Omron Sysmac Studio project Auto Connect Project (Sysmac Studio 1.45.1.64010, StandardProject)

# Controller new_Controller_0: NX102-9000 version 1.43
Units and slaves: Node1 : NX-ECC203 (E001); Unit 1 : NX-ID5342 (N1); Unit 2 : NX-ID5342 (N2); Unit 3 : NX-OD5121 (N3); Unit 4 : NX-OD5121 (N4); Node2 : NX-ECC203 (E002); Unit 1 : NX-ID5342 (N1_1); Unit 2 : NX-ID5342 (N2_1); Unit 3 : NX-OD5121 (N3_1); Unit 4 : NX-OD5121 (N4_1); Node3 : NX-ECC203 (E003); Unit 1 : NX-ID5342 (N5); Unit 2 : NX-ID5342 (N5_2); Unit 3 : NX-OD5121 (N6); Unit 4 : NX-OD5121 (N6_1); Node4 : NX-ECC203 (E004); Unit 1 : NX-ID5342 (N1_2); Unit 2 : NX-ID5342 (N2_2); Unit 3 : NX-OD5121 (N3_2); Unit 4 : NX-OD5121 (N4_2); Node5 : NX-ECC203 (E005); Unit 1 : NX-ID5342 (N7); Unit 2 : NX-ID5342 (N7_1); Unit 3 : NX-OD5121 (N8); Unit 4 : NX-OD5121 (N8_1); Node6 : NX-ECC203 (E006); Unit 1 : NX-ID5342 (N1_3); Unit 2 : NX-ID5342 (N2_3); Unit 3 : NX-OD5121 (N3_3); Unit 4 : NX-OD5121 (N4_3); Unit 1 : NX-PF0730 (N5_1); Unit 2 : NX-OD5121 (N3_6); Unit 3 : NX-ID5342 (N2_6)
Task PrimaryTask (priority 4, period or condition 2000): Program0

VAR_GLOBAL
    IN1_00 : BOOL;  (* at ECAT://node#[1,1]/Input Bit 16 bits/Input Bit 00 *)
    IN1_01 : BOOL;  (* at ECAT://node#[1,1]/Input Bit 16 bits/Input Bit 01 *)
    IN1_02 : BOOL;  (* at ECAT://node#[1,1]/Input Bit 16 bits/Input Bit 02 *)
    IN1_03 : BOOL;  (* at ECAT://node#[1,1]/Input Bit 16 bits/Input Bit 03 *)
    IN0_01 : BOOL;  (* PB RESET; at IOBus://unit#3/Input Bit 16 bits/Input Bit 01 *)
    IN0_00 : BOOL;  (* SS ENABLE; at IOBus://unit#3/Input Bit 16 bits/Input Bit 00 *)
    OUT100_00 : BOOL;  (* PL PLC RUN; at IOBus://unit#2/Output Bit 16 bits/Output Bit 00 *)
    OUT100_01 : BOOL;  (* PL FAULT; at IOBus://unit#2/Output Bit 16 bits/Output Bit 01 *)
    OUT100_02 : BOOL;  (* PL ENABLE MODE; at IOBus://unit#2/Output Bit 16 bits/Output Bit 02 *)
    OUT100_03 : BOOL;  (* PL KUNING; at IOBus://unit#2/Output Bit 16 bits/Output Bit 03 *)
    OUT100_04 : BOOL;  (* PL KUNING; at IOBus://unit#2/Output Bit 16 bits/Output Bit 04 *)
    OUT100_05 : BOOL;  (* BUZZER; at IOBus://unit#2/Output Bit 16 bits/Output Bit 05 *)
    OUT100_06 : BOOL;  (* TL RED; at IOBus://unit#2/Output Bit 16 bits/Output Bit 06 *)
    OUT100_07 : BOOL;  (* TL YELLOW; at IOBus://unit#2/Output Bit 16 bits/Output Bit 07 *)
    OUT100_08 : BOOL;  (* TL GREEN; at IOBus://unit#2/Output Bit 16 bits/Output Bit 08 *)
    OUT101_00 : BOOL;  (* FINISH PICK RACK 1; at ECAT://node#[1,3]/Output Bit 16 bits/Output Bit 00 *)
    OUT101_01 : BOOL;  (* at ECAT://node#[1,3]/Output Bit 16 bits/Output Bit 01 *)
    OUT101_02 : BOOL;  (* at ECAT://node#[1,3]/Output Bit 16 bits/Output Bit 02 *)
    OUT101_03 : BOOL;  (* at ECAT://node#[1,3]/Output Bit 16 bits/Output Bit 03 *)
    OUT101_04 : BOOL;  (* at ECAT://node#[1,3]/Output Bit 16 bits/Output Bit 04 *)
    OUT102_00 : BOOL;  (* at ECAT://node#[1,4]/Output Bit 16 bits/Output Bit 00 *)
    OUT103_00 : BOOL;  (* FINISH PICK RACK 2; at ECAT://node#[2,3]/Output Bit 16 bits/Output Bit 00 *)
    OUT103_01 : BOOL;  (* at ECAT://node#[2,3]/Output Bit 16 bits/Output Bit 01 *)
    OUT103_02 : BOOL;  (* at ECAT://node#[2,3]/Output Bit 16 bits/Output Bit 02 *)
    OUT103_03 : BOOL;  (* at ECAT://node#[2,3]/Output Bit 16 bits/Output Bit 03 *)
    OUT103_04 : BOOL;  (* at ECAT://node#[2,3]/Output Bit 16 bits/Output Bit 04 *)
    OUT103_05 : BOOL;  (* at ECAT://node#[2,3]/Output Bit 16 bits/Output Bit 05 *)
    OUT103_06 : BOOL;  (* at ECAT://node#[2,3]/Output Bit 16 bits/Output Bit 06 *)
    OUT103_07 : BOOL;  (* at ECAT://node#[2,3]/Output Bit 16 bits/Output Bit 07 *)
    OUT103_08 : BOOL;  (* at ECAT://node#[2,3]/Output Bit 16 bits/Output Bit 08 *)
    OUT103_09 : BOOL;  (* at ECAT://node#[2,3]/Output Bit 16 bits/Output Bit 09 *)
    OUT103_10 : BOOL;  (* at ECAT://node#[2,3]/Output Bit 16 bits/Output Bit 10 *)
    OUT104_00 : BOOL;  (* at ECAT://node#[2,4]/Output Bit 16 bits/Output Bit 00 *)
    OUT107_00 : BOOL;  (* at ECAT://node#[4,3]/Output Bit 16 bits/Output Bit 00 *)
    OUT107_01 : BOOL;  (* at ECAT://node#[4,3]/Output Bit 16 bits/Output Bit 01 *)
    OUT107_02 : BOOL;  (* at ECAT://node#[4,3]/Output Bit 16 bits/Output Bit 02 *)
    OUT107_03 : BOOL;  (* at ECAT://node#[4,3]/Output Bit 16 bits/Output Bit 03 *)
    OUT107_04 : BOOL;  (* at ECAT://node#[4,3]/Output Bit 16 bits/Output Bit 04 *)
    OUT107_05 : BOOL;  (* at ECAT://node#[4,3]/Output Bit 16 bits/Output Bit 05 *)
    OUT107_06 : BOOL;  (* at ECAT://node#[4,3]/Output Bit 16 bits/Output Bit 06 *)
    OUT107_07 : BOOL;  (* at ECAT://node#[4,3]/Output Bit 16 bits/Output Bit 07 *)
    OUT107_09 : BOOL;  (* at ECAT://node#[4,3]/Output Bit 16 bits/Output Bit 09 *)
    OUT107_10 : BOOL;  (* at ECAT://node#[4,3]/Output Bit 16 bits/Output Bit 10 *)
    OUT107_11 : BOOL;  (* at ECAT://node#[4,3]/Output Bit 16 bits/Output Bit 11 *)
    OUT107_12 : BOOL;  (* at ECAT://node#[4,3]/Output Bit 16 bits/Output Bit 12 *)
    OUT107_13 : BOOL;  (* at ECAT://node#[4,3]/Output Bit 16 bits/Output Bit 13 *)
    OUT107_14 : BOOL;  (* at ECAT://node#[4,3]/Output Bit 16 bits/Output Bit 14 *)
    OUT108_15 : BOOL;  (* at ECAT://node#[4,4]/Output Bit 16 bits/Output Bit 15 *)
    OUT111_01 : BOOL;  (* at ECAT://node#[6,3]/Output Bit 16 bits/Output Bit 01 *)
    OUT111_02 : BOOL;  (* at ECAT://node#[6,3]/Output Bit 16 bits/Output Bit 02 *)
    OUT112_00 : BOOL;  (* at ECAT://node#[6,4]/Output Bit 16 bits/Output Bit 00 *)
    OUT112_01 : BOOL;  (* at ECAT://node#[6,4]/Output Bit 16 bits/Output Bit 01 *)
    IN1_08 : BOOL;  (* at ECAT://node#[1,1]/Input Bit 16 bits/Input Bit 08 *)
    IN2_15 : BOOL;  (* at ECAT://node#[1,2]/Input Bit 16 bits/Input Bit 15 *)
    IN3_00 : BOOL;  (* at ECAT://node#[2,1]/Input Bit 16 bits/Input Bit 00 *)
    IN3_01 : BOOL;  (* at ECAT://node#[2,1]/Input Bit 16 bits/Input Bit 01 *)
    IN3_02 : BOOL;  (* at ECAT://node#[2,1]/Input Bit 16 bits/Input Bit 02 *)
    IN3_03 : BOOL;  (* at ECAT://node#[2,1]/Input Bit 16 bits/Input Bit 03 *)
    IN3_04 : BOOL;  (* at ECAT://node#[2,1]/Input Bit 16 bits/Input Bit 04 *)
    IN3_05 : BOOL;  (* at ECAT://node#[2,1]/Input Bit 16 bits/Input Bit 05 *)
    IN3_06 : BOOL;  (* at ECAT://node#[2,1]/Input Bit 16 bits/Input Bit 06 *)
    IN3_07 : BOOL;  (* at ECAT://node#[2,1]/Input Bit 16 bits/Input Bit 07 *)
    IN3_08 : BOOL;  (* at ECAT://node#[2,1]/Input Bit 16 bits/Input Bit 08 *)
    IN3_09 : BOOL;  (* at ECAT://node#[2,1]/Input Bit 16 bits/Input Bit 09 *)
    IN7_01 : BOOL;  (* at ECAT://node#[4,1]/Input Bit 16 bits/Input Bit 01 *)
    IN7_02 : BOOL;  (* at ECAT://node#[4,1]/Input Bit 16 bits/Input Bit 02 *)
    IN7_03 : BOOL;  (* at ECAT://node#[4,1]/Input Bit 16 bits/Input Bit 03 *)
    IN7_04 : BOOL;  (* at ECAT://node#[4,1]/Input Bit 16 bits/Input Bit 04 *)
    IN7_05 : BOOL;  (* at ECAT://node#[4,1]/Input Bit 16 bits/Input Bit 05 *)
    IN7_06 : BOOL;  (* at ECAT://node#[4,1]/Input Bit 16 bits/Input Bit 06 *)
    IN7_07 : BOOL;  (* at ECAT://node#[4,1]/Input Bit 16 bits/Input Bit 07 *)
    IN7_09 : BOOL;  (* at ECAT://node#[4,1]/Input Bit 16 bits/Input Bit 09 *)
    IN7_10 : BOOL;  (* at ECAT://node#[4,1]/Input Bit 16 bits/Input Bit 10 *)
    IN7_11 : BOOL;  (* at ECAT://node#[4,1]/Input Bit 16 bits/Input Bit 11 *)
    IN7_12 : BOOL;  (* at ECAT://node#[4,1]/Input Bit 16 bits/Input Bit 12 *)
    IN7_13 : BOOL;  (* at ECAT://node#[4,1]/Input Bit 16 bits/Input Bit 13 *)
    IN7_14 : BOOL;  (* at ECAT://node#[4,1]/Input Bit 16 bits/Input Bit 14 *)
    IN11_01 : BOOL;  (* at ECAT://node#[6,1]/Input Bit 16 bits/Input Bit 01 *)
    IN11_02 : BOOL;  (* at ECAT://node#[6,1]/Input Bit 16 bits/Input Bit 02 *)
    IN7_00 : BOOL;  (* at ECAT://node#[4,1]/Input Bit 16 bits/Input Bit 00 *)
    ATCO_NICKEL : BOOL;
    ATCO_LITHIUM : BOOL;
    NEW_BATTERY : BOOL;
    DATA_ATCO : WORD;  (* Area Loading *)
    PLC_ERROR_CODE : DWORD;
    OLD_DATA_ATCO : WORD;
    SEN_RACK1A_UP1 AT %W31.00 : BOOL;  (* published *)
    SEN_RACK1A_MD1 AT %W31.01 : BOOL;  (* published *)
    SEN_RACK1A_LO1 AT %W31.06 : BOOL;  (* published *)
    SEN_RACK1B_UP1 AT %W31.02 : BOOL;  (* published *)
    SEN_RACK1B_UP2 AT %W31.03 : BOOL;  (* published *)
    SEN_RACK1B_UP3 AT %W31.04 : BOOL;  (* published *)
    SEN_RACK1B_MD1 AT %W31.05 : BOOL;  (* published *)
    SEN_RACK1B_LO1 AT %W31.07 : BOOL;  (* published *)
    LAMP_RACK1A_UP1 AT %W21.00 : BOOL;  (* published *)
    LAMP_RACK1A_MD1 AT %W21.01 : BOOL;  (* published *)
    LAMP_RACK1A_LO1 AT %W21.06 : BOOL;  (* published *)
    LAMP_RACK1B_UP1 AT %W21.02 : BOOL;  (* published *)
    LAMP_RACK1B_UP2 AT %W21.03 : BOOL;  (* published *)
    LAMP_RACK1B_UP3 AT %W21.04 : BOOL;  (* published *)
    LAMP_RACK1B_MD1 AT %W21.05 : BOOL;  (* published *)
    LAMP_RACK1B_LO1 AT %W21.07 : BOOL;  (* published *)
    SEN_RACK2A_UP1 AT %W32.00 : BOOL;  (* published *)
    SEN_RACK2A_UP2 AT %W32.01 : BOOL;  (* published *)
    SEN_RACK2A_MD1 AT %W32.02 : BOOL;  (* published *)
    SEN_RACK2A_MD2 AT %W32.03 : BOOL;  (* published *)
    SEN_RACK2B_UP1 AT %W32.04 : BOOL;  (* published *)
    SEN_RACK2B_UP2 AT %W32.05 : BOOL;  (* published *)
    SEN_RACK2B_MD1 AT %W32.06 : BOOL;  (* published *)
    SEN_RACK2B_MD2 AT %W32.07 : BOOL;  (* published *)
    SEN_RACK2B_LO1 AT %W32.08 : BOOL;  (* published *)
    SEN_RACK2B_LO2 AT %W32.09 : BOOL;  (* published *)
    LAMP_RACK2A_UP1 AT %W22.00 : BOOL;  (* published *)
    LAMP_RACK2A_UP2 AT %W22.01 : BOOL;  (* published *)
    LAMP_RACK2A_MD1 AT %W22.02 : BOOL;  (* published *)
    LAMP_RACK2A_MD2 AT %W22.03 : BOOL;  (* published *)
    LAMP_RACK2B_UP1 AT %W22.04 : BOOL;  (* published *)
    LAMP_RACK2B_UP2 AT %W22.05 : BOOL;  (* published *)
    LAMP_RACK2B_MD1 AT %W22.06 : BOOL;  (* published *)
    LAMP_RACK2B_MD2 AT %W22.07 : BOOL;  (* published *)
    LAMP_RACK2B_LO1 AT %W22.08 : BOOL;  (* published *)
    LAMP_RACK2B_LO2 AT %W22.09 : BOOL;  (* published *)
    SEN_RACK3A_UP1 AT %W33.00 : BOOL;  (* published *)
    SEN_RACK3A_MD1 AT %W33.01 : BOOL;  (* published *)
    LAMP_RACK3A_UP1 AT %W23.00 : BOOL;  (* published *)
    LAMP_RACK3A_MD1 AT %W23.01 : BOOL;  (* published *)
    SEN_RACK4A_UP1 AT %W34.00 : BOOL;  (* published *)
    SEN_RACK4A_UP2 AT %W34.01 : BOOL;  (* published *)
    SEN_RACK4A_MD1 AT %W34.02 : BOOL;  (* published *)
    SEN_RACK4A_MD2 AT %W34.03 : BOOL;  (* published *)
    SEN_RACK4A_MD3 AT %W34.04 : BOOL;  (* published *)
    SEN_RACK4A_LO1 AT %W34.05 : BOOL;  (* published *)
    SEN_RACK4A_LO2 AT %W34.06 : BOOL;  (* published *)
    SEN_RACK4A_LO3 AT %W34.07 : BOOL;  (* published *)
    SEN_RACK4B_UP1 AT %W34.08 : BOOL;  (* published *)
    SEN_RACK4B_MD1 AT %W34.09 : BOOL;  (* published *)
    SEN_RACK4B_MD2 AT %W34.10 : BOOL;  (* published *)
    SEN_RACK4B_LO1 AT %W34.11 : BOOL;  (* published *)
    SEN_RACK4B_LO2 AT %W34.12 : BOOL;  (* published *)
    SEN_RACK4C_UP1 AT %W34.13 : BOOL;  (* published *)
    SEN_RACK4C_MD1 AT %W34.14 : BOOL;  (* published *)
    SEN_RACK4C_LO1 AT %W34.15 : BOOL;  (* published *)
    LAMP_RACK4A_UP1 AT %W24.00 : BOOL;  (* published *)
    LAMP_RACK4A_UP2 AT %W24.01 : BOOL;  (* published *)
    LAMP_RACK4A_MD1 AT %W24.02 : BOOL;  (* published *)
    LAMP_RACK4A_MD2 AT %W24.03 : BOOL;  (* published *)
    LAMP_RACK4A_MD3 AT %W24.04 : BOOL;  (* published *)
    LAMP_RACK4A_LO1 AT %W24.05 : BOOL;  (* published *)
    LAMP_RACK4A_LO2 AT %W24.06 : BOOL;  (* published *)
    LAMP_RACK4A_LO3 AT %W24.07 : BOOL;  (* published *)
    LAMP_RACK4B_UP1 AT %W24.08 : BOOL;  (* published *)
    LAMP_RACK4B_MD1 AT %W24.09 : BOOL;  (* published *)
    LAMP_RACK4B_MD2 AT %W24.10 : BOOL;  (* published *)
    LAMP_RACK4B_LO1 AT %W24.11 : BOOL;  (* published *)
    LAMP_RACK4B_LO2 AT %W24.12 : BOOL;  (* published *)
    LAMP_RACK4C_UP1 AT %W24.13 : BOOL;  (* published *)
    LAMP_RACK4C_MD1 AT %W24.14 : BOOL;  (* published *)
    LAMP_RACK4C_LO1 AT %W24.15 : BOOL;  (* published *)
    SEN_RACK5A_UP1 AT %W35.00 : BOOL;  (* published *)
    SEN_RACK5A_MD1 AT %W35.01 : BOOL;  (* published *)
    SEN_RACK5A_LO1 AT %W35.02 : BOOL;  (* published *)
    SEN_RACK5B_UP1 AT %W35.03 : BOOL;  (* published *)
    SEN_RACK5B_MD1 AT %W35.04 : BOOL;  (* published *)
    SEN_RACK5B_LO1 AT %W35.05 : BOOL;  (* published *)
    LAMP_RACK5A_UP1 AT %W25.00 : BOOL;  (* published *)
    LAMP_RACK5A_MD1 AT %W25.01 : BOOL;  (* published *)
    LAMP_RACK5A_LO1 AT %W25.02 : BOOL;  (* published *)
    LAMP_RACK5B_UP1 AT %W25.03 : BOOL;  (* published *)
    LAMP_RACK5B_MD1 AT %W25.04 : BOOL;  (* published *)
    LAMP_RACK5B_LO1 AT %W25.05 : BOOL;  (* published *)
    SEN_RACK6A_UP1 AT %W36.00 : BOOL;  (* published *)
    SEN_RACK6A_MD1 AT %W36.01 : BOOL;  (* published *)
    SEN_RACK6A_LO1 AT %W36.02 : BOOL;  (* published *)
    SEN_RACK6B_UP1 AT %W36.03 : BOOL;  (* published *)
    SEN_RACK6B_MD1 AT %W36.05 : BOOL;  (* published *)
    LAMP_RACK6A_UP1 AT %W26.00 : BOOL;  (* published *)
    LAMP_RACK6A_MD1 AT %W26.01 : BOOL;  (* published *)
    LAMP_RACK6A_LO1 AT %W26.02 : BOOL;  (* published *)
    LAMP_RACK6B_UP1 AT %W26.03 : BOOL;  (* published *)
    LAMP_RACK6B_MD1 AT %W26.05 : BOOL;  (* published *)
    SEN_RACK7A_UP1 AT %W37.00 : BOOL;  (* published *)
    SEN_RACK7B_UP1 AT %W37.01 : BOOL;  (* published *)
END_VAR
VAR_GLOBAL RETAIN
    TEACH_RACK1A_LO1 : WORD;
    TEACH_RACK1A_MD1 : WORD;
    TEACH_RACK1A_UP1 : WORD;
    TEACH_RACK1B_LO1 : WORD;
    TEACH_RACK1B_MD1 : WORD;
    TEACH_RACK1B_UP1 : WORD;
    TEACH_RACK1B_UP2 : WORD;
    TEACH_RACK1B_UP3 : WORD;
    TEACH_RACK2A_MD1 : WORD;
    TEACH_RACK2A_MD2 : WORD;
    TEACH_RACK2A_UP1 : WORD;
    TEACH_RACK2A_UP2 : WORD;
    TEACH_RACK2B_LO1 : WORD;
    TEACH_RACK2B_LO2 : WORD;
    TEACH_RACK2B_MD1 : WORD;
    TEACH_RACK2B_MD2 : WORD;
    TEACH_RACK2B_UP1 : WORD;
    TEACH_RACK2B_UP2 : WORD;
    TEACH_RACK3A_MD1 : WORD;
    TEACH_RACK3A_UP1 : WORD;
    TEACH_RACK4A_LO1 : WORD;
    TEACH_RACK4A_LO2 : WORD;
    TEACH_RACK4A_LO3 : WORD;
    TEACH_RACK4A_MD1 : WORD;
    TEACH_RACK4A_MD2 : WORD;
    TEACH_RACK4A_MD3 : WORD;
    TEACH_RACK4A_UP1 : WORD;
    TEACH_RACK4A_UP2 : WORD;
    TEACH_RACK4B_LO1 : WORD;
    TEACH_RACK4B_LO2 : WORD;
    TEACH_RACK4B_MD1 : WORD;
    TEACH_RACK4B_MD2 : WORD;
    TEACH_RACK4B_UP1 : WORD;
    TEACH_RACK4C_LO1 : WORD;
    TEACH_RACK4C_MD1 : WORD;
    TEACH_RACK4C_UP1 : WORD;
    TEACH_RACK5A_LO1 : WORD;
    TEACH_RACK5A_MD1 : WORD;
    TEACH_RACK5A_UP1 : WORD;
    TEACH_RACK5B_LO1 : WORD;
    TEACH_RACK5B_MD1 : WORD;
    TEACH_RACK5B_UP1 : WORD;
    TEACH_RACK6A_LO1 : WORD;
    TEACH_RACK6A_MD1 : WORD;
    TEACH_RACK6A_UP1 : WORD;
    TEACH_RACK6B_MD1 : WORD;
    TEACH_RACK6B_UP1 : WORD;
    TEACH_RACK7A_UP1 : WORD;
END_VAR
VAR_GLOBAL
    LAMP_RACK7A_UP1 AT %W27.00 : BOOL;  (* published *)
    LAMP_RACK7B_UP1 AT %W27.01 : BOOL;  (* published *)
    FINISH_PICK_RACK1 : BOOL;
    FINISH_PICK_RACK2 : BOOL;
    FINISH_PICK_RACK4 : BOOL;
    FINISH_PICK_RACK6 : BOOL;
    FINISH_PICK_RACK7 : BOOL;
    FAULT_PICK_FALSE_RACK1 : BOOL;
    FAULT_PICK_FALSE_RACK2 : BOOL;
    FAULT_PICK_FALSE_RACK4 : BOOL;
    FAULT_PICK_FALSE_RACK6 : BOOL;
    FAULT_PICK_FALSE_RACK7 : BOOL;
    FAULT_PICK_TOO_MUCH_RACK1 : BOOL;
    FAULT_PICK_TOO_MUCH_RACK2 : BOOL;
    FAULT_PICK_TOO_MUCH_RACK4 : BOOL;
    FAULT_PICK_TOO_MUCH_RACK6 : BOOL;
    FAULT_PICK_TOO_MUCH_RACK7 : BOOL;
END_VAR
VAR_GLOBAL RETAIN
    TEACH_RACK7B_UP1 : WORD;
END_VAR
VAR_GLOBAL
    ATCO_UDP_CONNECTED : BOOL;
    DATA_ATCO_1 : WORD;  (* Area Lower Case *)
    DATA_ATCO_2 : WORD;  (* Area BBM *)
    DATA_ATCO_3 : WORD;  (* Area Manual Tightening *)
    DATA_ATCO_4 : WORD;  (* Area Charging *)
    ATCO_NICKEL_1 : BOOL;
    ATCO_LITHIUM_1 : BOOL;
    NEW_BATTERY_1 : BOOL;
    ATCO_NICKEL_2 : BOOL;
    ATCO_LITHIUM_2 : BOOL;
    NEW_BATTERY_2 : BOOL;
    ATCO_NICKEL_3 : BOOL;
    ATCO_LITHIUM_3 : BOOL;
    NEW_BATTERY_3 : BOOL;
    ATCO_NICKEL_4 : BOOL;
    ATCO_LITHIUM_4 : BOOL;
    NEW_BATTERY_4 : BOOL;
    FLAG_ERROR_PICK : BOOL;
END_VAR
VAR_GLOBAL RETAIN
    HMI_SET_1A_UP1 AT %D0 : INT;  (* published *)
    HMI_SET_1A_MD1 AT %D1 : INT;  (* published *)
    HMI_SET_1B_UP1 AT %D2 : INT;  (* published *)
    HMI_SET_1B_UP2 AT %D3 : INT;  (* published *)
    HMI_SET_1B_UP3 AT %D4 : INT;  (* published *)
    HMI_SET_1B_MD1 AT %D5 : INT;  (* published *)
    HMI_SET_2A_UP1 AT %D6 : INT;  (* published *)
    HMI_SET_2A_UP2 AT %D7 : INT;  (* published *)
    HMI_SET_2A_MD1 AT %D8 : INT;  (* published *)
    HMI_SET_2A_MD2 AT %D9 : INT;  (* published *)
    HMI_SET_2B_UP1 AT %D10 : INT;  (* published *)
    HMI_SET_2B_UP2 AT %D11 : INT;  (* published *)
    HMI_SET_2B_MD1 AT %D12 : INT;  (* published *)
    HMI_SET_2B_MD2 AT %D13 : INT;  (* published *)
    HMI_SET_2B_LO1 AT %D14 : INT;  (* published *)
    HMI_SET_2B_LO2 AT %D15 : INT;  (* published *)
    HMI_SET_3A_UP1 AT %D16 : INT;  (* published *)
    HMI_SET_3A_MD1 AT %D17 : INT;  (* published *)
    HMI_SET_4A_UP1 AT %D18 : INT;  (* published *)
    HMI_SET_4A_UP2 AT %D19 : INT;  (* published *)
    HMI_SET_4A_MD1 AT %D20 : INT;  (* published *)
    HMI_SET_4A_MD2 AT %D21 : INT;  (* published *)
    HMI_SET_4A_MD3 AT %D22 : INT;  (* published *)
    HMI_SET_4A_LO1 AT %D23 : INT;  (* published *)
    HMI_SET_4A_LO2 AT %D24 : INT;  (* published *)
    HMI_SET_4A_LO3 AT %D25 : INT;  (* published *)
    HMI_SET_4B_UP1 AT %D26 : INT;  (* published *)
    HMI_SET_4B_MD1 AT %D27 : INT;  (* published *)
    HMI_SET_4B_MD2 AT %D28 : INT;  (* published *)
    HMI_SET_4B_LO1 AT %D29 : INT;  (* published *)
    HMI_SET_4B_LO2 AT %D30 : INT;  (* published *)
    HMI_SET_4C_UP1 AT %D31 : INT;  (* published *)
    HMI_SET_4C_MD1 AT %D32 : INT;  (* published *)
    HMI_SET_4C_LO1 AT %D33 : INT;  (* published *)
    HMI_SET_5A_UP1 AT %D34 : INT;  (* published *)
    HMI_SET_5A_MD1 AT %D35 : INT;  (* published *)
    HMI_SET_5A_LO1 AT %D36 : INT;  (* published *)
    HMI_SET_5B_UP1 AT %D37 : INT;  (* published *)
    HMI_SET_5B_MD1 AT %D38 : INT;  (* published *)
    HMI_SET_6A_UP1 AT %D39 : INT;  (* published *)
    HMI_SET_6A_MD1 AT %D40 : INT;  (* published *)
    HMI_SET_6A_LO1 AT %D41 : INT;  (* published *)
    HMI_SET_6B_UP1 AT %D42 : INT;  (* published *)
    HMI_SET_6B_UP2 AT %D43 : INT;  (* published *)
    HMI_SET_6B_MD1 AT %D44 : INT;  (* published *)
END_VAR
VAR_GLOBAL
    HMI_POWER_ON AT %W0.08 : BOOL;  (* published *)
    HMI_ENABLE AT %W0.01 : BOOL;  (* published *)
    HMI_CONNECT AT %W0.02 : BOOL;  (* published *)
    HMI_NICKEL_BATTERY AT %W0.03 : BOOL;  (* published *)
    HMI_LITHIUM_BATTERY AT %W0.04 : BOOL;  (* published *)
    HMI_PLC_RUN AT %W0.05 : BOOL;  (* published *)
    HMI_FAULT AT %W0.06 : BOOL;  (* published *)
    HMI_ENABLE_SETTING AT %W0.07 : BOOL;  (* published *)
    HMI_LAMPU_1A_UP1 AT %W1.00 : BOOL;  (* published *)
    HMI_LAMPU_1A_MD1 AT %W1.01 : BOOL;  (* published *)
    HMI_LAMPU_1B_UP1 AT %W1.02 : BOOL;  (* published *)
    HMI_LAMPU_1B_UP2 AT %W1.03 : BOOL;  (* published *)
    HMI_LAMPU_1B_UP3 AT %W1.04 : BOOL;  (* published *)
    HMI_LAMPU_1B_MD1 AT %W1.05 : BOOL;  (* published *)
    HMI_LAMPU_2A_UP1 AT %W2.00 : BOOL;  (* published *)
    HMI_LAMPU_2A_UP2 AT %W2.01 : BOOL;  (* published *)
    HMI_LAMPU_2A_MD1 AT %W2.02 : BOOL;  (* published *)
    HMI_LAMPU_2A_MD2 AT %W2.03 : BOOL;  (* published *)
    HMI_LAMPU_2B_UP1 AT %W2.04 : BOOL;  (* published *)
    HMI_LAMPU_2B_UP2 AT %W2.05 : BOOL;  (* published *)
    HMI_LAMPU_2B_MD1 AT %W2.06 : BOOL;  (* published *)
    HMI_LAMPU_2B_MD2 AT %W2.07 : BOOL;  (* published *)
    HMI_LAMPU_2B_LO1 AT %W2.08 : BOOL;  (* published *)
    HMI_LAMPU_2B_LO2 AT %W2.09 : BOOL;  (* published *)
    HMI_LAMPU_3A_UP1 AT %W3.00 : BOOL;  (* published *)
    HMI_LAMPU_3A_MD1 AT %W3.01 : BOOL;  (* published *)
    HMI_LAMPU_4A_UP1 AT %W4.00 : BOOL;  (* published *)
    HMI_LAMPU_4A_UP2 AT %W4.01 : BOOL;  (* published *)
    HMI_LAMPU_4A_MD1 AT %W4.02 : BOOL;  (* published *)
    HMI_LAMPU_4A_MD2 AT %W4.03 : BOOL;  (* published *)
    HMI_LAMPU_4A_MD3 AT %W4.04 : BOOL;  (* published *)
    HMI_LAMPU_4A_LO1 AT %W4.05 : BOOL;  (* published *)
    HMI_LAMPU_4A_LO2 AT %W4.06 : BOOL;  (* published *)
    HMI_LAMPU_4A_LO3 AT %W4.07 : BOOL;  (* published *)
    HMI_LAMPU_4B_UP1 AT %W4.08 : BOOL;  (* published *)
    HMI_LAMPU_4B_MD1 AT %W4.09 : BOOL;  (* published *)
    HMI_LAMPU_4B_MD2 AT %W4.10 : BOOL;  (* published *)
    HMI_LAMPU_4B_LO1 AT %W4.11 : BOOL;  (* published *)
    HMI_LAMPU_4B_LO2 AT %W4.12 : BOOL;  (* published *)
    HMI_LAMPU_4C_UP1 AT %W4.13 : BOOL;  (* published *)
    HMI_LAMPU_4C_MD1 AT %W4.14 : BOOL;  (* published *)
    HMI_LAMPU_4C_LO1 AT %W4.15 : BOOL;  (* published *)
    HMI_LAMPU_5A_UP1 AT %W5.00 : BOOL;  (* published *)
    HMI_LAMPU_5A_MD1 AT %W5.01 : BOOL;  (* published *)
    HMI_LAMPU_5A_LO1 AT %W5.02 : BOOL;  (* published *)
    HMI_LAMPU_5B_UP1 AT %W5.03 : BOOL;  (* published *)
    HMI_LAMPU_5B_MD1 AT %W5.04 : BOOL;  (* published *)
    HMI_LAMPU_6A_UP1 AT %W6.00 : BOOL;  (* published *)
    HMI_LAMPU_6A_MD1 AT %W6.01 : BOOL;  (* published *)
    HMI_LAMPU_6A_LO1 AT %W6.02 : BOOL;  (* published *)
    HMI_LAMPU_6B_UP1 AT %W6.03 : BOOL;  (* published *)
    HMI_LAMPU_6B_UP2 AT %W6.04 : BOOL;  (* published *)
    HMI_LAMPU_6B_MD1 AT %W6.05 : BOOL;  (* published *)
END_VAR
VAR_GLOBAL RETAIN
    TEACH_RACK6B_UP2 : WORD;
END_VAR
VAR_GLOBAL
    RECIEVECJ_DONE : BOOL;
    HMI_LAMPU_1A_UP2 AT %W1.06 : BOOL;  (* published *)
    HMI_LAMPU_1A_UP3 AT %W1.07 : BOOL;  (* published *)
    HMI_LAMPU_3A_UP2 AT %W3.02 : BOOL;  (* published *)
    HMI_LAMPU_3A_UP3 AT %W3.03 : BOOL;  (* published *)
    HMI_LAMPU_3A_MD2 AT %W3.04 : BOOL;  (* published *)
    HMI_LAMPU_7A_UP1 AT %W7.00 : BOOL;
    HMI_LAMPU_7A_UP2 AT %W7.01 : BOOL;
END_VAR
VAR_GLOBAL RETAIN
    HMI_SET_7A_UP1 AT %D45 : INT;  (* published *)
    HMI_SET_7A_UP2 AT %D46 : INT;  (* published *)
    HMI_SET_3A_UP2 AT %D47 : INT;  (* published *)
    HMI_SET_3A_UP3 AT %D48 : INT;  (* published *)
    HMI_SET_3A_MD2 AT %D49 : INT;  (* published *)
    HMI_SET_1A_UP2 AT %D50 : INT;  (* published *)
    HMI_SET_1A_UP3 AT %D51 : INT;  (* published *)
END_VAR
VAR_GLOBAL
    HMI_BATTERY_SETTING AT %W0.00 : BOOL;  (* published *)
    WAIT_ALARM : BOOL;
    BUZZER_OFF AT %W0.09 : BOOL;  (* published *)
END_VAR
VAR_GLOBAL RETAIN
    RAK_1_CONDITION AT %D47 : INT;  (* published *)
    RAK_2_CONDITION AT %D48 : INT;  (* published *)
    RAK_3_CONDITION AT %D49 : INT;  (* published *)
    RAK_4_CONDITION AT %D50 : INT;  (* published *)
    RAK_5_CONDITION AT %D51 : INT;  (* published *)
    RAK_6_CONDITION AT %D52 : INT;  (* published *)
    RAK_7_CONDITION AT %D53 : INT;  (* published *)
END_VAR
VAR_GLOBAL
    HMI_FAULT_PICKING AT %W0.10 : BOOL;  (* published *)
    HMI_FAULT_WAIT_PICKING AT %W0.11 : BOOL;  (* published *)
    HMI_FAULT_CONNECTION AT %W0.12 : BOOL;  (* published *)
    PROX_SUB_CONVEYOR_1 : BOOL;
    HMI_RESET_CJ AT %W0.13 : BOOL;  (* published *)
    HMI_FORCE_RAK_1 AT %W10.00 : BOOL;  (* published *)
    HMI_FORCE_RAK_2 AT %W10.01 : BOOL;  (* published *)
    HMI_FORCE_RAK_3 AT %W10.02 : BOOL;  (* published *)
    HMI_FORCE_RAK_4 AT %W10.03 : BOOL;  (* published *)
    HMI_FORCE_RAK_5 AT %W10.04 : BOOL;  (* published *)
    HMI_FORCE_RAK_6 AT %W10.05 : BOOL;  (* published *)
    HMI_FORCE_RAK_7 AT %W10.06 : BOOL;  (* published *)
    HMI_ENABLE_SWITCH AT %W0.14 : BOOL;  (* published *)
    HMI_RESET_BUTTON AT %W0.15 : BOOL;  (* published *)
    HMI_EC_NODE_1_ERR AT %W90.00 : BOOL;
    HMI_EC_NODE_2_ERR AT %W90.01 : BOOL;
    HMI_EC_NODE_3_ERR AT %W90.02 : BOOL;
    HMI_EC_NODE_4_ERR AT %W90.03 : BOOL;
    HMI_PLC_ERROR AT %W91.00 : BOOL;
    SEN_RACK4A_LO4 AT %W35.06 : BOOL;
    LAMP_RACK4A_LO4 AT %W25.06 : BOOL;
    HMI_LAMPU_4A_LO4 AT %W5.06 : BOOL;
END_VAR
VAR_GLOBAL RETAIN
    HMI_SET_4A_LO4 AT %D54 : INT;
END_VAR
VAR_GLOBAL
    TEACH_RACK4A_LO4 : WORD;
END_VAR
VAR_GLOBAL CONSTANT
    NX3 : _sNXUNIT_ID := (NodeAdr := 3, IPAdr := [5(16#FF)], UnitNo := 0, Path := [16#11, 16#0, 16#2, 16#0, 16#3, 16#0, 16#1, 16#0, 16#2, 55(16#0)], PathLength := 12);  (* NODE 3 *)
END_VAR

PROGRAM Program0
VAR
    ENABLE_MODE : BOOL;
    FLAG_FAULT : BOOL;
    PLC_ERROR : BOOL;
    RESET_PLC_ERROR : BOOL;
    ResetPLCError0 : ResetPLCError;
    PICKING_SEQ_RACK_1 : FB_PICKING_SEQ;
    PICKING_SEQ_RACK_2 : FB_PICKING_SEQ;
    PICKING_SEQ_RACK_4 : FB_PICKING_SEQ;
    PICKING_SEQ_RACK_6 : FB_PICKING_SEQ;
    PICKING_SEQ_RACK_7 : FB_PICKING_SEQ;
    TON_ATCO_FINISH_RACK_1 : TON;  (* ' *)
    RESET_ATCO_FINISH_PICK_RACK_1 : BOOL;
    RESET_ATCO_FINISH_PICK_RACK_2 : BOOL;
    TON_ATCO_FINISH_RACK_2 : TON;
    RESET_ATCO_FINISH_PICK_RACK_4 : BOOL;
    TON_ATCO_FINISH_RACK_4 : TON;
    RESET_ATCO_FINISH_PICK_RACK_6 : BOOL;
    TON_ATCO_FINISH_RACK_6 : TON;
    CREATE_UDP_SOCKET_ATCO : SktUDPCreate;
    CONNECTING_ATCO : BOOL;
    ERROR_CREATE_UDP_ATCO : BOOL;
    RECONNECTING_ATCO : BOOL;
    RECEIVE_UDP_SOCKET_ATCO : SktUDPRcv;
    ERROR_RECEIVE_UDP_ATCO : BOOL;
    ATCO_UDP_DISCONNECTED : BOOL;
    ATCO_UDP_DATA_RECEIVED : BOOL;
    SOCKET_ATCO : _sSOCKET;
    IpAdr : STRING[256] := '192.168.4.111';
    PortNo : UINT := 9600;
    ATCO_UDP_DATA : ARRAY[0..98] OF BYTE;
    SEND_UDP_SOCKET_ATCO : SktUDPSend;
    ERROR_SEND_UDP_ATCO : BOOL;
    RESET_BYTE : ARRAY[0..98] OF BYTE;
    ATCO_UDP_DATA_SENT : BOOL;
    CLOSE_UDP_SOCKET_ATCO : SktClose;
    pseudo_reset : BOOL;
    test : BOOL;
    data1 : UDINT;
    data2 : UINT;
    data3 : STRING[255];
    data4 : STRING[255];
    data5 : UINT;
    coba : BOOL;
    busy1 : BOOL;
    error1 : WORD;
    online : BOOL;
    test1 : BOOL;
    busy2 : BOOL;
    error2 : WORD;
    test2 : BOOL;
    data6 : UINT;
    socket1 : _sSOCKET_ADDRESS;
    NetAdr : _sDNET_ADR := (NetNo := 0, NodeNo := 111, UnitNo := 16#0);
    recieve_cj : Rcv;
    recieve_dat : ARRAY[0..1] OF WORD;
    option : _sRESPONSE := (isNonResp := False, TimeOut := 10, Retry := 1);
    busy_risif : BOOL;
    error_risif : BOOL;
    errorid_risif : WORD;
    erroridex_risif : DWORD;
    recieve_dat1 : ARRAY[0..1] OF WORD;
    recieve_dat2 : ARRAY[0..1] OF WORD;
    recieve_dat3 : ARRAY[0..1] OF WORD;
    RESET_ENABLE : BOOL;
    recieve_cj2 : Rcv;
    recieve_cj3 : Rcv;
    p : BOOL;
    TIM_ENABLE : BOOL;
    timer_on_enable : _sTimer;
    recieve_dat4 : ARRAY[0..1] OF WORD;
    hmi1 : BOOL;
    recieve_cj4 : Rcv;
    recieve_cj5 : Rcv;
    FAULT_PICK_TOO_MUCH_RACK3 : BOOL;
    PSEUDO_FINISH_PICK_2 : BOOL;
    FINISH_PICK_RACK3 : BOOL;
    FINISH_PICK_RACK5 : BOOL;
    PSEUDO_ON : TON;
    COBA1 : BOOL;
    busy_risif_2 : BOOL;
    error_risif_2 : BOOL;
    errorid_risif_2 : WORD;
    erroridex_risif_2 : DWORD;
    busy_risif_1 : BOOL;
    error_risif_1 : BOOL;
    errorid_risif_1 : WORD;
    erroridex_risif_1 : DWORD;
    busy_risif_3 : BOOL;
    error_risif_3 : BOOL;
    errorid_risif_3 : WORD;
    erroridex_risif_3 : DWORD;
    busy_risif_4 : BOOL;
    error_risif_4 : BOOL;
    errorid_risif_4 : WORD;
    erroridex_risif_4 : DWORD;
    TIMER_PICK_TOO_LONG : TON;
    ET_PICK_LONG : TIME;
    RST_TIM_RAK_1 : BOOL;
    RST_TIM_RAK_2 : BOOL;
    RST_TIM_RAK_4 : BOOL;
    RST_TIM_RAK_6 : BOOL;
    RST_TIM_RAK_7 : BOOL;
    ERROR_ID_CONNECTION : BOOL;
    ERROR_IDEX_CONNECTION : BOOL;
    TIM_BUSY : TON;
    TIM_BUSY_1 : TON;
    TIM_BUSY_2 : TON;
    TIM_BUSY_3 : TON;
    TIM_BUSY_4 : TON;
    BUSY_CONNECTION : BOOL;
    TIMER_PICK_TOO_LONG_1 : TON;
    TIMER_PICK_TOO_LONG_2 : TON;
    ET_PICK_LONG_1 : TIME;
    ET_PICK_LONG_2 : TIME;
    TRTIAL1 : BOOL;
    TRTIAL2 : BOOL;
    RETRY_CJ : BOOL;
    TIM_RETRY_CJ : TON;
    FLAG_CJ_ERROR : BOOL;
    TIM_ERROR_CJ : TON;
    TIMER_RST_RAK1 : TON;
    TIMER_RST_RAK2 : TON;
    TIMER_RST_RAK4 : TON;
    TIMER_RST_RAK6 : TON;
    TIMER_RST_RAK7 : TON;
    PROX_SUB_CONVEYOR_1 : BOOL;
    SEND_CJ : Send;
    busy_send : BOOL;
    error_send : BOOL;
    errorid_send : WORD;
    erroridex_send : DWORD;
    SEND_CJ_DAT : ARRAY[0..1] OF WORD;
    SEND_CJ_2 : Send;
    SEND_CJ_DAT_2 : ARRAY[0..1] OF WORD;
    busy_send_2 : BOOL;
    error_send_2 : BOOL;
    errorid_send_2 : WORD;
    erroridex_send_2 : DWORD;
    SEND_CJ_3 : Send;
    SEND_CJ_DAT_3 : ARRAY[0..1] OF WORD;
    busy_send_3 : BOOL;
    error_send_3 : BOOL;
    errorid_send_3 : WORD;
    erroridex_send_3 : DWORD;
    SEND_CJ_4 : Send;
    SEND_CJ_DAT_4 : ARRAY[0..1] OF WORD;
    error_send_4 : BOOL;
    errorid_send_4 : WORD;
    erroridex_send_4 : DWORD;
    SEND_CJ_5 : Send;
    busy_send_4 : BOOL;
    SEND_CJ_DAT_5 : ARRAY[0..1] OF WORD;
    busy_send_5 : BOOL;
    error_send_5 : BOOL;
    errorid_send_5 : WORD;
    erroridex_send_5 : DWORD;
    RETRY_CJ_1 : BOOL;
    RETRY_CJ_2 : BOOL;
    RETRY_CJ_3 : BOOL;
    RETRY_CJ_4 : BOOL;
    HMI : BOOL;
    TON_RETRY_CJ : TON;
    ET_RETRY_CJ : TIME;
    TON_RECEIVE_CJ : TON;
    TON_RECEIVE_CJ2 : TON;
    ET_RETRY_CJ2 : TIME;
    TON_RETRY_CJ2 : TON;
    TON_RECEIVE_CJ3 : TON;
    ET_RETRY_CJ3 : TIME;
    TON_RETRY_CJ3 : TON;
    TON_RECEIVE_CJ1 : TON;
    ET_RETRY_CJ1 : TIME;
    TON_RETRY_CJ1 : TON;
    TON_RETRY_CJ4 : TON;
    ET_RETRY_CJ4 : TIME;
    TON_RECEIVE_CJ4 : TON;
    ResetECError1 : ResetECError;
    _EC : BOOL;
    RESTART_NX3 : RestartNXUnit;
    ET_TIMER_RST_RAK1 : TIME;
    ET_TIMER_RST_RAK2 : TIME;
    ET_TIMER_RST_RAK4 : TIME;
    ET_TIMER_RST_RAK6 : TIME;
    ET_TIMER_RST_RAK7 : TIME;
END_VAR
VAR_EXTERNAL
    OUT100_00 : BOOL;
    IN0_00 : BOOL;
    OUT100_03 : BOOL;
    OUT100_02 : BOOL;  (* FAULT LAMP *)
    OUT100_01 : BOOL;  (* PL_ENABLE *)
    OUT100_04 : BOOL;
    OUT100_05 : BOOL;  (* Buzzer *)
    IN0_01 : BOOL;
    OUT100_07 : BOOL;  (* TL YELLOW *)
    OUT100_06 : BOOL;  (* TL RED *)
    NEW_BATTERY : BOOL;
    DATA_ATCO : WORD;
    ATCO_NICKEL : BOOL;
    ATCO_LITHIUM : BOOL;
    PLC_ERROR_CODE : DWORD;
    OLD_DATA_ATCO : WORD;
    OUT108_15 : BOOL;
    SEN_RACK1A_LO1 : BOOL;
    IN1_00 : BOOL;
    SEN_RACK1A_MD1 : BOOL;
    SEN_RACK1A_UP1 : BOOL;
    SEN_RACK1B_LO1 : BOOL;
    SEN_RACK1B_MD1 : BOOL;
    SEN_RACK1B_UP1 : BOOL;
    SEN_RACK1B_UP2 : BOOL;
    SEN_RACK1B_UP3 : BOOL;
    SEN_RACK2A_MD1 : BOOL;
    SEN_RACK2A_MD2 : BOOL;
    SEN_RACK2A_UP1 : BOOL;
    SEN_RACK2A_UP2 : BOOL;
    SEN_RACK2B_LO1 : BOOL;
    SEN_RACK2B_LO2 : BOOL;
    SEN_RACK2B_MD1 : BOOL;
    SEN_RACK2B_MD2 : BOOL;
    SEN_RACK2B_UP1 : BOOL;
    SEN_RACK2B_UP2 : BOOL;
    SEN_RACK3A_MD1 : BOOL;
    SEN_RACK4A_LO1 : BOOL;
    SEN_RACK4A_LO2 : BOOL;
    SEN_RACK4A_LO3 : BOOL;
    SEN_RACK4A_MD1 : BOOL;
    SEN_RACK4A_MD2 : BOOL;
    SEN_RACK4A_MD3 : BOOL;
    SEN_RACK4A_UP1 : BOOL;
    SEN_RACK4A_UP2 : BOOL;
    SEN_RACK4B_LO1 : BOOL;
    SEN_RACK4B_LO2 : BOOL;
    SEN_RACK4B_MD1 : BOOL;
    SEN_RACK4B_MD2 : BOOL;
    SEN_RACK4B_UP1 : BOOL;
    SEN_RACK4C_LO1 : BOOL;
    SEN_RACK4C_MD1 : BOOL;
    SEN_RACK4C_UP1 : BOOL;
    SEN_RACK6A_LO1 : BOOL;
    SEN_RACK6A_MD1 : BOOL;
    SEN_RACK6A_UP1 : BOOL;
    SEN_RACK6B_MD1 : BOOL;
    SEN_RACK6B_UP1 : BOOL;
    SEN_RACK7A_UP1 : BOOL;
    SEN_RACK7B_UP1 : BOOL;
    LAMP_RACK1A_LO1 : BOOL;
    OUT101_01 : BOOL;
    LAMP_RACK1A_MD1 : BOOL;
    LAMP_RACK1A_UP1 : BOOL;
    LAMP_RACK1B_LO1 : BOOL;
    LAMP_RACK1B_MD1 : BOOL;
    LAMP_RACK1B_UP1 : BOOL;
    LAMP_RACK1B_UP2 : BOOL;
    LAMP_RACK1B_UP3 : BOOL;
    LAMP_RACK2A_MD1 : BOOL;
    LAMP_RACK2A_MD2 : BOOL;
    LAMP_RACK2A_UP1 : BOOL;
    LAMP_RACK2A_UP2 : BOOL;
    LAMP_RACK2B_LO1 : BOOL;
    LAMP_RACK2B_LO2 : BOOL;
    LAMP_RACK2B_MD1 : BOOL;
    LAMP_RACK2B_MD2 : BOOL;
    LAMP_RACK2B_UP1 : BOOL;
    LAMP_RACK2B_UP2 : BOOL;
    LAMP_RACK4A_LO1 : BOOL;
    LAMP_RACK4A_LO2 : BOOL;
    LAMP_RACK4A_LO3 : BOOL;
    LAMP_RACK4A_MD1 : BOOL;
    LAMP_RACK4A_MD2 : BOOL;
    LAMP_RACK4A_MD3 : BOOL;
    LAMP_RACK4A_UP1 : BOOL;
    LAMP_RACK4A_UP2 : BOOL;
    LAMP_RACK4B_LO1 : BOOL;
    LAMP_RACK4B_LO2 : BOOL;
    LAMP_RACK4B_MD1 : BOOL;
    LAMP_RACK4B_MD2 : BOOL;
    LAMP_RACK4B_UP1 : BOOL;
    LAMP_RACK4C_LO1 : BOOL;
    LAMP_RACK4C_MD1 : BOOL;
    LAMP_RACK4C_UP1 : BOOL;
    LAMP_RACK5A_LO1 : BOOL;
    LAMP_RACK6A_LO1 : BOOL;
    LAMP_RACK6A_MD1 : BOOL;
    LAMP_RACK6A_UP1 : BOOL;
    LAMP_RACK6B_MD1 : BOOL;
    LAMP_RACK6B_UP1 : BOOL;
    LAMP_RACK7A_UP1 : BOOL;
    LAMP_RACK7B_UP1 : BOOL;
    FINISH_PICK_RACK1 : BOOL;
    FAULT_PICK_FALSE_RACK1 : BOOL;
    FAULT_PICK_TOO_MUCH_RACK1 : BOOL;
    TEACH_RACK1A_UP1 : WORD;
    TEACH_RACK1B_UP2 : WORD;
    TEACH_RACK1B_UP1 : WORD;
    TEACH_RACK1B_UP3 : WORD;
    TEACH_RACK1B_MD1 : WORD;
    OUT101_00 : BOOL;
    FINISH_PICK_RACK2 : BOOL;
    OUT103_00 : BOOL;
    FAULT_PICK_FALSE_RACK2 : BOOL;
    FAULT_PICK_TOO_MUCH_RACK2 : BOOL;
    TEACH_RACK2A_UP1 : WORD;
    TEACH_RACK2A_UP2 : WORD;
    TEACH_RACK2A_MD1 : WORD;
    TEACH_RACK2A_MD2 : WORD;
    TEACH_RACK2B_UP1 : WORD;
    TEACH_RACK2B_UP2 : WORD;
    TEACH_RACK2B_MD1 : WORD;
    TEACH_RACK2B_MD2 : WORD;
    TEACH_RACK2B_LO1 : WORD;
    TEACH_RACK2B_LO2 : WORD;
    FINISH_PICK_RACK4 : BOOL;
    FAULT_PICK_FALSE_RACK4 : BOOL;
    FAULT_PICK_TOO_MUCH_RACK4 : BOOL;
    FINISH_PICK_RACK6 : BOOL;
    FAULT_PICK_FALSE_RACK6 : BOOL;
    FAULT_PICK_TOO_MUCH_RACK6 : BOOL;
    TEACH_RACK6B_MD1 : WORD;
    FINISH_PICK_RACK7 : BOOL;
    FAULT_PICK_FALSE_RACK7 : BOOL;
    FAULT_PICK_TOO_MUCH_RACK7 : BOOL;
    TEACH_RACK7B_UP1 : WORD;
    TEACH_RACK4A_UP1 : WORD;
    TEACH_RACK4A_UP2 : WORD;
    TEACH_RACK4A_MD1 : WORD;
    TEACH_RACK4A_MD2 : WORD;
    TEACH_RACK4A_MD3 : WORD;
    TEACH_RACK4A_LO1 : WORD;
    TEACH_RACK4A_LO2 : WORD;
    TEACH_RACK4A_LO3 : WORD;
    TEACH_RACK4B_MD1 : WORD;
    TEACH_RACK4B_MD2 : WORD;
    TEACH_RACK4B_LO1 : WORD;
    TEACH_RACK4B_LO2 : WORD;
    IN1_03 : BOOL;
    IN1_02 : BOOL;
    IN1_01 : BOOL;
    IN3_07 : BOOL;
    IN3_06 : BOOL;
    IN3_03 : BOOL;
    IN3_02 : BOOL;
    IN3_09 : BOOL;
    IN1_08 : BOOL;
    IN3_08 : BOOL;
    IN3_05 : BOOL;
    IN3_04 : BOOL;
    IN3_01 : BOOL;
    IN3_00 : BOOL;
    IN7_13 : BOOL;
    IN7_12 : BOOL;
    IN7_11 : BOOL;
    IN7_07 : BOOL;
    IN7_06 : BOOL;
    IN7_05 : BOOL;
    IN7_01 : BOOL;
    IN7_00 : BOOL;
    IN7_10 : BOOL;
    IN7_09 : BOOL;
    IN7_02 : BOOL;
    IN7_03 : BOOL;
    IN7_04 : BOOL;
    IN11_02 : BOOL;
    IN11_01 : BOOL;
    OUT101_04 : BOOL;
    OUT101_03 : BOOL;
    OUT101_02 : BOOL;
    OUT103_08 : BOOL;
    OUT103_07 : BOOL;
    OUT103_04 : BOOL;
    OUT103_03 : BOOL;
    OUT103_10 : BOOL;
    OUT103_09 : BOOL;
    OUT103_06 : BOOL;
    OUT103_05 : BOOL;
    OUT103_02 : BOOL;
    OUT103_01 : BOOL;
    OUT107_13 : BOOL;
    OUT107_12 : BOOL;
    OUT107_11 : BOOL;
    OUT107_07 : BOOL;
    OUT107_06 : BOOL;
    OUT107_05 : BOOL;
    OUT107_01 : BOOL;
    OUT107_02 : BOOL;
    OUT107_00 : BOOL;
    OUT107_10 : BOOL;
    OUT107_09 : BOOL;
    OUT107_04 : BOOL;
    OUT107_03 : BOOL;
    OUT111_01 : BOOL;
    OUT111_02 : BOOL;
    TEACH_RACK4C_MD1 : WORD;
    OUT102_00 : BOOL;  (* ATCO FINISH PICK RACK 1 *)
    OUT104_00 : BOOL;  (* ATCO FINISH PICK RACK 2 *)
    OUT112_00 : BOOL;  (* ATCO FINISH PICK RACK 4 *)
    OUT112_01 : BOOL;  (* ATCO FINISH PICK RACK 6 *)
    ATCO_UDP_CONNECTED : BOOL;
END_VAR
VAR_EXTERNAL CONSTANT
    _EIP_EtnOnlineSta : BOOL;
    _EIP2_EtnOnlineSta : BOOL;
END_VAR
VAR_EXTERNAL
    DATA_ATCO_1 : WORD;
    DATA_ATCO_2 : WORD;
    DATA_ATCO_3 : WORD;
    ATCO_NICKEL_1 : BOOL;
    ATCO_LITHIUM_1 : BOOL;
    NEW_BATTERY_1 : BOOL;
    ATCO_NICKEL_2 : BOOL;
    ATCO_LITHIUM_2 : BOOL;
    NEW_BATTERY_2 : BOOL;
    ATCO_NICKEL_3 : BOOL;
    ATCO_LITHIUM_3 : BOOL;
    NEW_BATTERY_3 : BOOL;
    ATCO_LITHIUM_4 : BOOL;
    ATCO_NICKEL_4 : BOOL;
    DATA_ATCO_4 : WORD;
    NEW_BATTERY_4 : BOOL;
    FLAG_ERROR_PICK : BOOL;
    HMI_POWER_ON : BOOL;
    HMI_PLC_RUN : BOOL;
    HMI_ENABLE : BOOL;
    HMI_FAULT : BOOL;
    HMI_LAMPU_1B_MD1 : BOOL;
    HMI_LAMPU_1B_UP1 : BOOL;
    HMI_LAMPU_1B_UP2 : BOOL;
    HMI_LAMPU_1B_UP3 : BOOL;
    HMI_LAMPU_2A_MD1 : BOOL;
    HMI_LAMPU_2A_MD2 : BOOL;
    HMI_LAMPU_2A_UP1 : BOOL;
    HMI_LAMPU_2A_UP2 : BOOL;
    HMI_LAMPU_2B_LO1 : BOOL;
    HMI_LAMPU_2B_LO2 : BOOL;
    HMI_LAMPU_2B_MD1 : BOOL;
    HMI_LAMPU_2B_MD2 : BOOL;
    HMI_LAMPU_2B_UP1 : BOOL;
    HMI_LAMPU_2B_UP2 : BOOL;
    HMI_LAMPU_4A_LO1 : BOOL;
    HMI_LAMPU_4A_LO2 : BOOL;
    HMI_LAMPU_4A_LO3 : BOOL;
    HMI_LAMPU_4A_MD1 : BOOL;
    HMI_LAMPU_4A_MD2 : BOOL;
    HMI_LAMPU_4A_MD3 : BOOL;
    HMI_LAMPU_4A_UP1 : BOOL;
    HMI_LAMPU_4A_UP2 : BOOL;
    HMI_LAMPU_4B_LO1 : BOOL;
    HMI_LAMPU_4B_LO2 : BOOL;
    HMI_LAMPU_4B_MD1 : BOOL;
    HMI_LAMPU_4B_MD2 : BOOL;
    HMI_LAMPU_4C_MD1 : BOOL;
    HMI_LAMPU_6B_MD1 : BOOL;
    HMI_LAMPU_1A_MD1 : BOOL;
    HMI_SET_1A_MD1 : INT;
    HMI_ENABLE_SETTING : BOOL;
    TEACH_RACK1A_MD1 : WORD;
    HMI_SET_1A_UP1 : INT;
    TEACH_RACK1A_LO1 : WORD;
    HMI_SET_1B_UP1 : INT;
    HMI_SET_1B_UP2 : INT;
    HMI_SET_1B_UP3 : INT;
    HMI_SET_1B_MD1 : INT;
    HMI_SET_2A_UP1 : INT;
    HMI_SET_2A_UP2 : INT;
    HMI_SET_2A_MD1 : INT;
    HMI_SET_2A_MD2 : INT;
    HMI_SET_2B_UP1 : INT;
    HMI_SET_2B_UP2 : INT;
    HMI_SET_2B_MD1 : INT;
    HMI_SET_2B_MD2 : INT;
    HMI_SET_2B_LO1 : INT;
    HMI_SET_2B_LO2 : INT;
    HMI_SET_3A_UP1 : INT;
    HMI_SET_3A_MD1 : INT;
    HMI_SET_4A_UP1 : INT;
    HMI_SET_4A_UP2 : INT;
    HMI_SET_4A_MD1 : INT;
    HMI_SET_4A_MD2 : INT;
    HMI_SET_4A_MD3 : INT;
    HMI_SET_4A_LO1 : INT;
    HMI_SET_4A_LO2 : INT;
    HMI_SET_4A_LO3 : INT;
    HMI_SET_4B_UP1 : INT;
    HMI_SET_4B_MD1 : INT;
    HMI_SET_4B_MD2 : INT;
    HMI_SET_4B_LO1 : INT;
    HMI_SET_4B_LO2 : INT;
    HMI_SET_4C_UP1 : INT;
    HMI_SET_4C_MD1 : INT;
    HMI_SET_4C_LO1 : INT;
    HMI_SET_5A_UP1 : INT;
    HMI_SET_5A_MD1 : INT;
    HMI_SET_5A_LO1 : INT;
    HMI_SET_5B_UP1 : INT;
    HMI_SET_5B_MD1 : INT;
    HMI_SET_6A_UP1 : INT;
    HMI_SET_6A_MD1 : INT;
    HMI_SET_6A_LO1 : INT;
    HMI_SET_6B_MD1 : INT;
    HMI_SET_6B_UP1 : INT;
    HMI_SET_6B_UP2 : INT;
    TEACH_RACK3A_UP1 : WORD;
    TEACH_RACK3A_MD1 : WORD;
    TEACH_RACK4B_UP1 : WORD;
    TEACH_RACK4C_UP1 : WORD;
    TEACH_RACK4C_LO1 : WORD;
    TEACH_RACK5A_UP1 : WORD;
    TEACH_RACK5A_MD1 : WORD;
    TEACH_RACK5A_LO1 : WORD;
    TEACH_RACK5B_UP1 : WORD;
    TEACH_RACK5B_MD1 : WORD;
    TEACH_RACK6A_UP1 : WORD;
    TEACH_RACK6A_MD1 : WORD;
    TEACH_RACK6A_LO1 : WORD;
    TEACH_RACK6B_UP1 : WORD;
    TEACH_RACK6B_UP2 : WORD;
    RECIEVECJ_DONE : BOOL;
    HMI_CONNECT : BOOL;
    HMI_NICKEL_BATTERY : BOOL;
    HMI_LITHIUM_BATTERY : BOOL;
    OUT100_08 : BOOL;
    HMI_SET_7A_UP1 : INT;
    HMI_BATTERY_SETTING : BOOL;
    WAIT_ALARM : BOOL;
    BUZZER_OFF : BOOL;
    RAK_1_CONDITION : INT;
    RAK_2_CONDITION : INT;
    RAK_4_CONDITION : INT;
    RAK_6_CONDITION : INT;
    RAK_7_CONDITION : INT;
    HMI_FAULT_PICKING : BOOL;
    HMI_FAULT_WAIT_PICKING : BOOL;
    HMI_FAULT_CONNECTION : BOOL;
    HMI_LAMPU_7A_UP1 : BOOL;
    IN2_15 : BOOL;
    HMI_RESET_CJ : BOOL;
    HMI_FORCE_RAK_1 : BOOL;
    HMI_FORCE_RAK_2 : BOOL;
    HMI_FORCE_RAK_3 : BOOL;
    HMI_FORCE_RAK_4 : BOOL;
    HMI_FORCE_RAK_5 : BOOL;
    HMI_FORCE_RAK_6 : BOOL;
    HMI_FORCE_RAK_7 : BOOL;
    HMI_ENABLE_SWITCH : BOOL;
    HMI_RESET_BUTTON : BOOL;
END_VAR
VAR_EXTERNAL CONSTANT
    _EC_DisconnSlavTbl : ARRAY[1..192] OF BOOL;
    _EC_CommErrTbl : ARRAY[1..192] OF BOOL;
    _EC_PDSlavTbl : ARRAY[1..192] OF BOOL;
END_VAR
VAR_EXTERNAL
    HMI_EC_NODE_1_ERR : BOOL;
    HMI_EC_NODE_2_ERR : BOOL;
    HMI_EC_NODE_3_ERR : BOOL;
    HMI_EC_NODE_4_ERR : BOOL;
    HMI_PLC_ERROR : BOOL;
    IN7_14 : BOOL;
    SEN_RACK4A_LO4 : BOOL;
    OUT107_14 : BOOL;
    LAMP_RACK4A_LO4 : BOOL;
    HMI_LAMPU_4A_LO4 : BOOL;
    HMI_SET_4A_LO4 : INT;
    TEACH_RACK4A_LO4 : WORD;
END_VAR
VAR_EXTERNAL CONSTANT
    NX3 : _sNXUNIT_ID;
END_VAR
VAR
    _t1 : BOOL;
    _t2 : BOOL;
    _p3 : BOOL;
    _e4 : R_TRIG;
    _e5 : R_TRIG;
    _e6 : R_TRIG;
    _e7 : R_TRIG;
    _e8 : R_TRIG;
    _e9 : R_TRIG;
    _e10 : R_TRIG;
    _e11 : R_TRIG;
    _e12 : R_TRIG;
    _e13 : R_TRIG;
    _e14 : R_TRIG;
    _e15 : R_TRIG;
    _e16 : R_TRIG;
    _e17 : R_TRIG;
    _e18 : R_TRIG;
    _e19 : R_TRIG;
    _e20 : R_TRIG;
    _e21 : R_TRIG;
    _e22 : R_TRIG;
    _e23 : R_TRIG;
    _e24 : R_TRIG;
    _e25 : R_TRIG;
    _e26 : R_TRIG;
    _e27 : R_TRIG;
    _e28 : R_TRIG;
    _e29 : R_TRIG;
    _e30 : R_TRIG;
    _e31 : R_TRIG;
    _e32 : R_TRIG;
    _e33 : R_TRIG;
    _e34 : R_TRIG;
    _e35 : R_TRIG;
    _e36 : R_TRIG;
    _e37 : R_TRIG;
    _e38 : R_TRIG;
    _e39 : R_TRIG;
    _e40 : R_TRIG;
    _e41 : R_TRIG;
    _e42 : R_TRIG;
    _e43 : R_TRIG;
    _e44 : R_TRIG;
    _e45 : R_TRIG;
    _e46 : R_TRIG;
    _e47 : R_TRIG;
    _e48 : R_TRIG;
    _e49 : R_TRIG;
    _e50 : R_TRIG;
    _e51 : R_TRIG;
    _e52 : R_TRIG;
    _e53 : R_TRIG;
END_VAR

(* Section MAIN_PROGRAM: ladder, written here as Structured Text *)

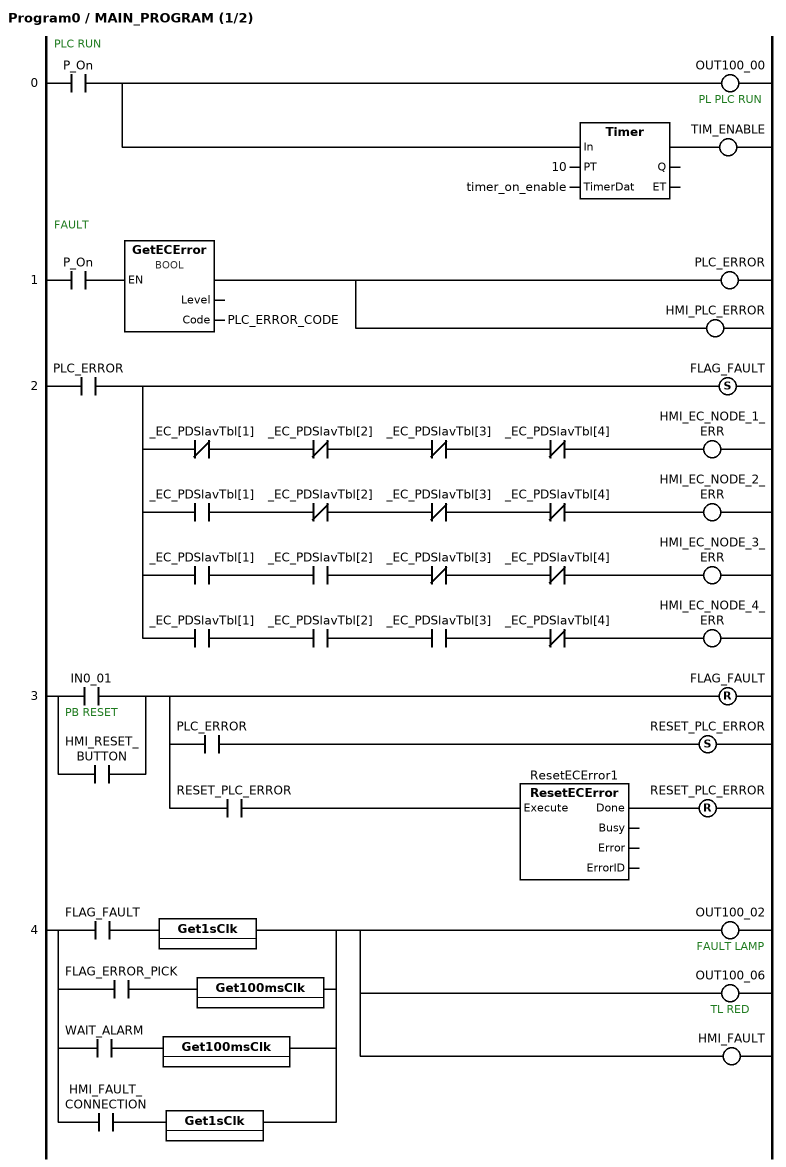
(* Rung 0: PLC RUN *)
OUT100_00 := P_On;
_t1 := Timer(In := P_On, PT := 10, TimerDat := timer_on_enable);
TIM_ENABLE := _t1;
(* Rung 1: FAULT *)
_t2 := FALSE;
IF P_On THEN _t2 := GetECError(Code => PLC_ERROR_CODE); END_IF;
PLC_ERROR := _t2;
HMI_PLC_ERROR := _t2;
(* Rung 2 *)
IF PLC_ERROR THEN FLAG_FAULT := TRUE; END_IF;
HMI_EC_NODE_1_ERR := PLC_ERROR AND NOT _EC_PDSlavTbl[1] AND NOT _EC_PDSlavTbl[2] AND NOT _EC_PDSlavTbl[3] AND NOT _EC_PDSlavTbl[4];
HMI_EC_NODE_2_ERR := PLC_ERROR AND _EC_PDSlavTbl[1] AND NOT _EC_PDSlavTbl[2] AND NOT _EC_PDSlavTbl[3] AND NOT _EC_PDSlavTbl[4];
HMI_EC_NODE_3_ERR := PLC_ERROR AND _EC_PDSlavTbl[1] AND _EC_PDSlavTbl[2] AND NOT _EC_PDSlavTbl[3] AND NOT _EC_PDSlavTbl[4];
HMI_EC_NODE_4_ERR := PLC_ERROR AND _EC_PDSlavTbl[1] AND _EC_PDSlavTbl[2] AND _EC_PDSlavTbl[3] AND NOT _EC_PDSlavTbl[4];
(* Rung 3 *)
IF IN0_01 OR HMI_RESET_BUTTON THEN FLAG_FAULT := FALSE; END_IF;
IF (IN0_01 OR HMI_RESET_BUTTON) AND PLC_ERROR THEN RESET_PLC_ERROR := TRUE; END_IF;
ResetECError1(Execute := (IN0_01 OR HMI_RESET_BUTTON) AND RESET_PLC_ERROR);
IF ResetECError1.Done THEN RESET_PLC_ERROR := FALSE; END_IF;
(* Rung 4 *)
_p3 := (FLAG_FAULT AND Get1sClk()) OR (FLAG_ERROR_PICK AND Get100msClk()) OR (WAIT_ALARM AND Get100msClk()) OR (HMI_FAULT_CONNECTION AND Get1sClk());
OUT100_02 := _p3;
OUT100_06 := _p3;
HMI_FAULT := _p3;

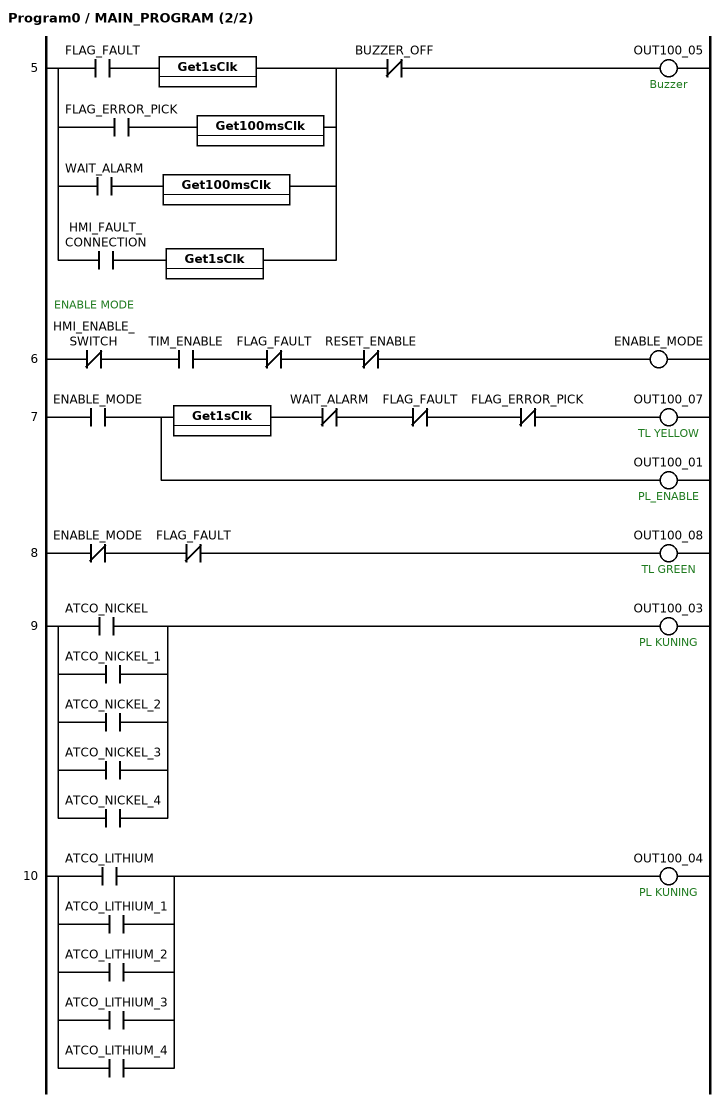
(* Rung 5 *)
OUT100_05 := ((FLAG_FAULT AND Get1sClk()) OR (FLAG_ERROR_PICK AND Get100msClk()) OR (WAIT_ALARM AND Get100msClk()) OR (HMI_FAULT_CONNECTION AND Get1sClk())) AND NOT BUZZER_OFF;
(* Rung 6: ENABLE MODE *)
ENABLE_MODE := NOT HMI_ENABLE_SWITCH AND TIM_ENABLE AND NOT FLAG_FAULT AND NOT RESET_ENABLE;
(* Rung 7 *)
OUT100_07 := ENABLE_MODE AND Get1sClk() AND NOT WAIT_ALARM AND NOT FLAG_FAULT AND NOT FLAG_ERROR_PICK;
OUT100_01 := ENABLE_MODE;
(* Rung 8 *)
OUT100_08 := NOT ENABLE_MODE AND NOT FLAG_FAULT;
(* Rung 9 *)
OUT100_03 := ATCO_NICKEL OR ATCO_NICKEL_1 OR ATCO_NICKEL_2 OR ATCO_NICKEL_3 OR ATCO_NICKEL_4;
(* Rung 10 *)
OUT100_04 := ATCO_LITHIUM OR ATCO_LITHIUM_1 OR ATCO_LITHIUM_2 OR ATCO_LITHIUM_3 OR ATCO_LITHIUM_4;

(* Section HMI: ladder, written here as Structured Text *)

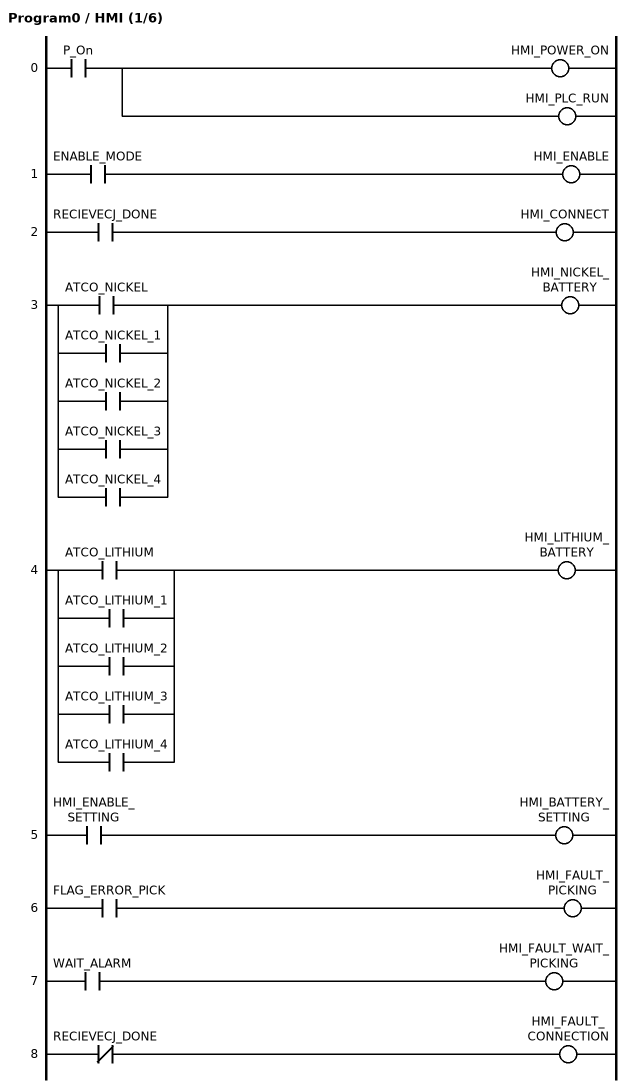
(* Rung 0 *)
HMI_POWER_ON := P_On;
HMI_PLC_RUN := P_On;
(* Rung 1 *)
HMI_ENABLE := ENABLE_MODE;
(* Rung 2 *)
HMI_CONNECT := RECIEVECJ_DONE;
(* Rung 3 *)
HMI_NICKEL_BATTERY := ATCO_NICKEL OR ATCO_NICKEL_1 OR ATCO_NICKEL_2 OR ATCO_NICKEL_3 OR ATCO_NICKEL_4;
(* Rung 4 *)
HMI_LITHIUM_BATTERY := ATCO_LITHIUM OR ATCO_LITHIUM_1 OR ATCO_LITHIUM_2 OR ATCO_LITHIUM_3 OR ATCO_LITHIUM_4;
(* Rung 5 *)
HMI_BATTERY_SETTING := HMI_ENABLE_SETTING;
(* Rung 6 *)
HMI_FAULT_PICKING := FLAG_ERROR_PICK;
(* Rung 7 *)
HMI_FAULT_WAIT_PICKING := WAIT_ALARM;
(* Rung 8 *)
HMI_FAULT_CONNECTION := NOT RECIEVECJ_DONE;

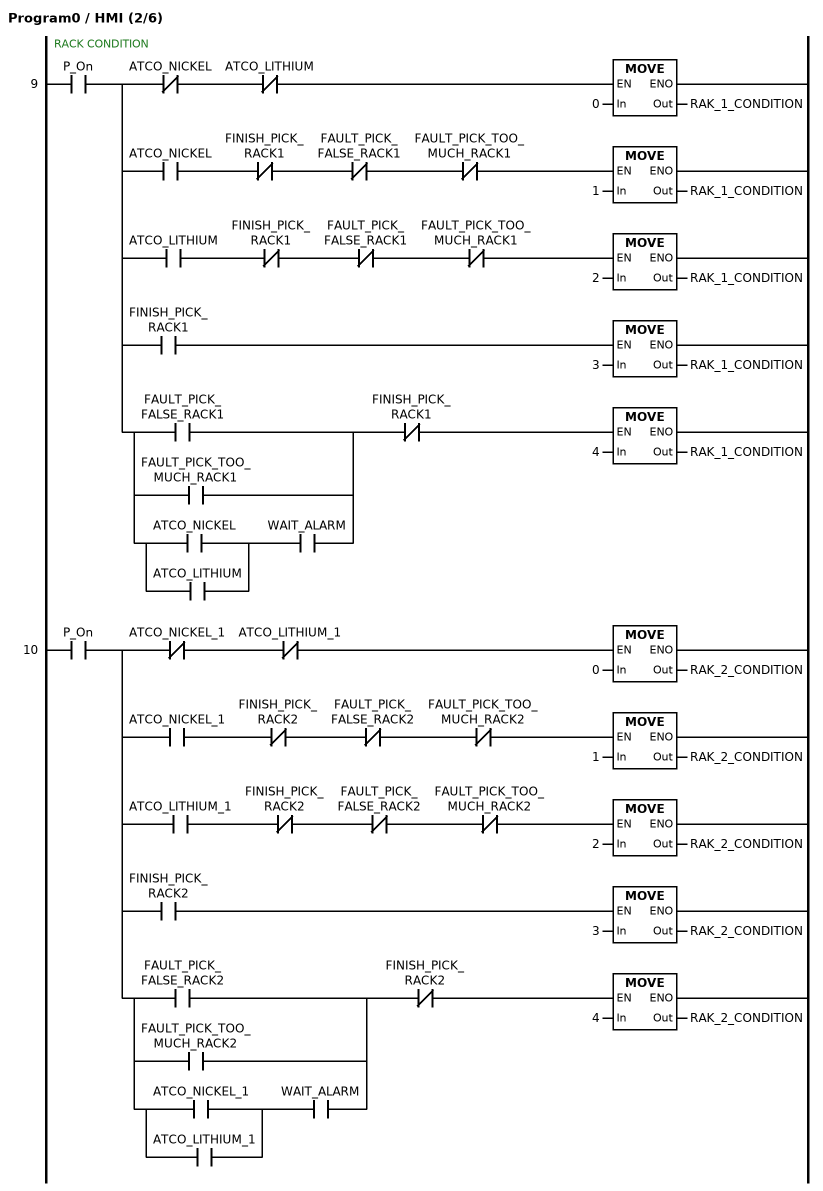
(* Rung 9: RACK CONDITION *)
IF P_On AND NOT ATCO_NICKEL AND NOT ATCO_LITHIUM THEN RAK_1_CONDITION := 0; END_IF;
IF P_On AND ATCO_NICKEL AND NOT FINISH_PICK_RACK1 AND NOT FAULT_PICK_FALSE_RACK1 AND NOT FAULT_PICK_TOO_MUCH_RACK1 THEN
    RAK_1_CONDITION := 1;
END_IF;
IF P_On AND ATCO_LITHIUM AND NOT FINISH_PICK_RACK1 AND NOT FAULT_PICK_FALSE_RACK1 AND NOT FAULT_PICK_TOO_MUCH_RACK1 THEN
    RAK_1_CONDITION := 2;
END_IF;
IF P_On AND FINISH_PICK_RACK1 THEN RAK_1_CONDITION := 3; END_IF;
IF P_On AND (FAULT_PICK_FALSE_RACK1 OR FAULT_PICK_TOO_MUCH_RACK1 OR ((ATCO_NICKEL OR ATCO_LITHIUM) AND WAIT_ALARM)) AND NOT FINISH_PICK_RACK1 THEN
    RAK_1_CONDITION := 4;
END_IF;
(* Rung 10 *)
IF P_On AND NOT ATCO_NICKEL_1 AND NOT ATCO_LITHIUM_1 THEN RAK_2_CONDITION := 0; END_IF;
IF P_On AND ATCO_NICKEL_1 AND NOT FINISH_PICK_RACK2 AND NOT FAULT_PICK_FALSE_RACK2 AND NOT FAULT_PICK_TOO_MUCH_RACK2 THEN
    RAK_2_CONDITION := 1;
END_IF;
IF P_On AND ATCO_LITHIUM_1 AND NOT FINISH_PICK_RACK2 AND NOT FAULT_PICK_FALSE_RACK2 AND NOT FAULT_PICK_TOO_MUCH_RACK2 THEN
    RAK_2_CONDITION := 2;
END_IF;
IF P_On AND FINISH_PICK_RACK2 THEN RAK_2_CONDITION := 3; END_IF;
IF P_On AND (FAULT_PICK_FALSE_RACK2 OR FAULT_PICK_TOO_MUCH_RACK2 OR ((ATCO_NICKEL_1 OR ATCO_LITHIUM_1) AND WAIT_ALARM)) AND NOT FINISH_PICK_RACK2 THEN
    RAK_2_CONDITION := 4;
END_IF;

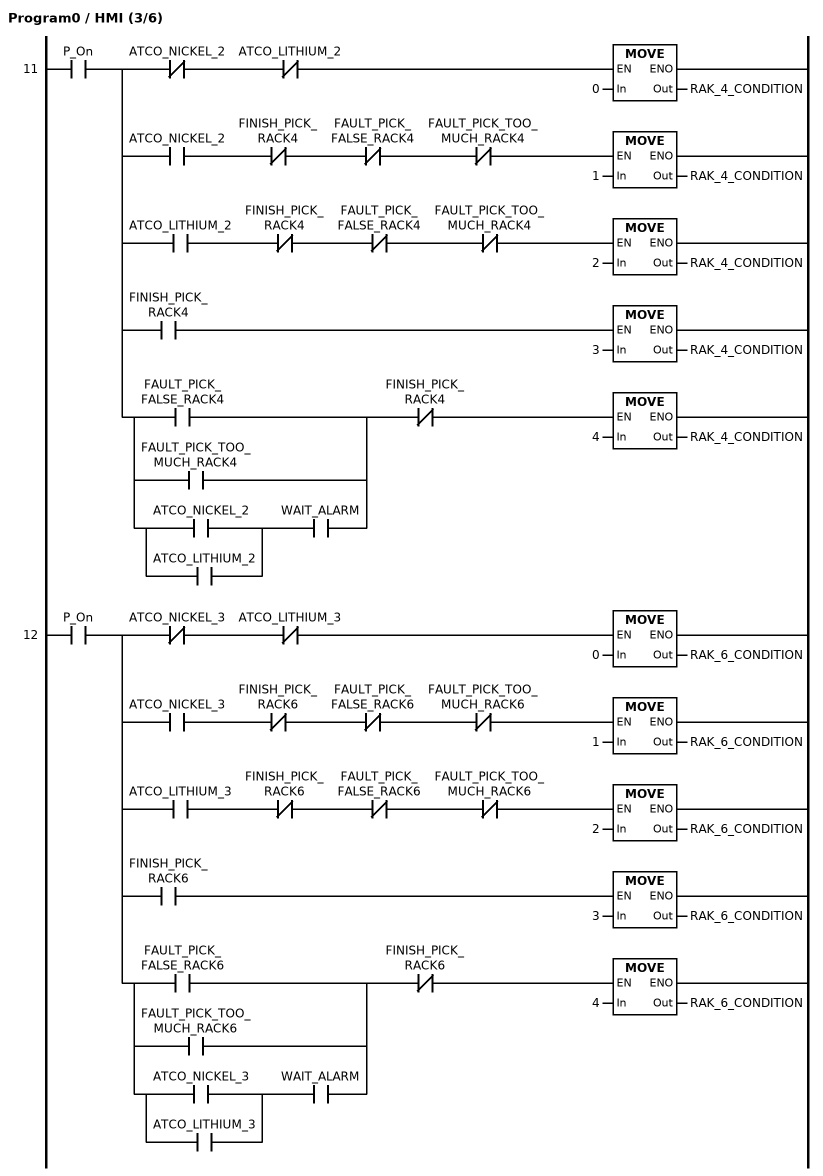
(* Rung 11 *)
IF P_On AND NOT ATCO_NICKEL_2 AND NOT ATCO_LITHIUM_2 THEN RAK_4_CONDITION := 0; END_IF;
IF P_On AND ATCO_NICKEL_2 AND NOT FINISH_PICK_RACK4 AND NOT FAULT_PICK_FALSE_RACK4 AND NOT FAULT_PICK_TOO_MUCH_RACK4 THEN
    RAK_4_CONDITION := 1;
END_IF;
IF P_On AND ATCO_LITHIUM_2 AND NOT FINISH_PICK_RACK4 AND NOT FAULT_PICK_FALSE_RACK4 AND NOT FAULT_PICK_TOO_MUCH_RACK4 THEN
    RAK_4_CONDITION := 2;
END_IF;
IF P_On AND FINISH_PICK_RACK4 THEN RAK_4_CONDITION := 3; END_IF;
IF P_On AND (FAULT_PICK_FALSE_RACK4 OR FAULT_PICK_TOO_MUCH_RACK4 OR ((ATCO_NICKEL_2 OR ATCO_LITHIUM_2) AND WAIT_ALARM)) AND NOT FINISH_PICK_RACK4 THEN
    RAK_4_CONDITION := 4;
END_IF;
(* Rung 12 *)
IF P_On AND NOT ATCO_NICKEL_3 AND NOT ATCO_LITHIUM_3 THEN RAK_6_CONDITION := 0; END_IF;
IF P_On AND ATCO_NICKEL_3 AND NOT FINISH_PICK_RACK6 AND NOT FAULT_PICK_FALSE_RACK6 AND NOT FAULT_PICK_TOO_MUCH_RACK6 THEN
    RAK_6_CONDITION := 1;
END_IF;
IF P_On AND ATCO_LITHIUM_3 AND NOT FINISH_PICK_RACK6 AND NOT FAULT_PICK_FALSE_RACK6 AND NOT FAULT_PICK_TOO_MUCH_RACK6 THEN
    RAK_6_CONDITION := 2;
END_IF;
IF P_On AND FINISH_PICK_RACK6 THEN RAK_6_CONDITION := 3; END_IF;
IF P_On AND (FAULT_PICK_FALSE_RACK6 OR FAULT_PICK_TOO_MUCH_RACK6 OR ((ATCO_NICKEL_3 OR ATCO_LITHIUM_3) AND WAIT_ALARM)) AND NOT FINISH_PICK_RACK6 THEN
    RAK_6_CONDITION := 4;
END_IF;

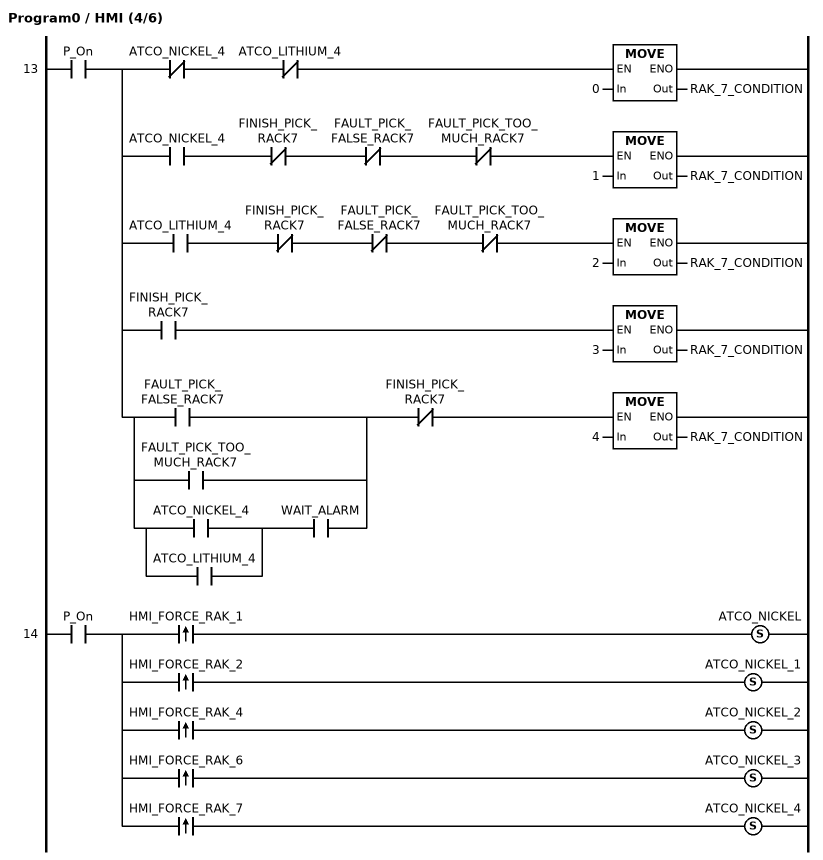
(* Rung 13 *)
IF P_On AND NOT ATCO_NICKEL_4 AND NOT ATCO_LITHIUM_4 THEN RAK_7_CONDITION := 0; END_IF;
IF P_On AND ATCO_NICKEL_4 AND NOT FINISH_PICK_RACK7 AND NOT FAULT_PICK_FALSE_RACK7 AND NOT FAULT_PICK_TOO_MUCH_RACK7 THEN
    RAK_7_CONDITION := 1;
END_IF;
IF P_On AND ATCO_LITHIUM_4 AND NOT FINISH_PICK_RACK7 AND NOT FAULT_PICK_FALSE_RACK7 AND NOT FAULT_PICK_TOO_MUCH_RACK7 THEN
    RAK_7_CONDITION := 2;
END_IF;
IF P_On AND FINISH_PICK_RACK7 THEN RAK_7_CONDITION := 3; END_IF;
IF P_On AND (FAULT_PICK_FALSE_RACK7 OR FAULT_PICK_TOO_MUCH_RACK7 OR ((ATCO_NICKEL_4 OR ATCO_LITHIUM_4) AND WAIT_ALARM)) AND NOT FINISH_PICK_RACK7 THEN
    RAK_7_CONDITION := 4;
END_IF;
(* Rung 14 *)
_e4(CLK := HMI_FORCE_RAK_1);
IF P_On AND _e4.Q THEN ATCO_NICKEL := TRUE; END_IF;
_e5(CLK := HMI_FORCE_RAK_2);
IF P_On AND _e5.Q THEN ATCO_NICKEL_1 := TRUE; END_IF;
_e6(CLK := HMI_FORCE_RAK_4);
IF P_On AND _e6.Q THEN ATCO_NICKEL_2 := TRUE; END_IF;
_e7(CLK := HMI_FORCE_RAK_6);
IF P_On AND _e7.Q THEN ATCO_NICKEL_3 := TRUE; END_IF;
_e8(CLK := HMI_FORCE_RAK_7);
IF P_On AND _e8.Q THEN ATCO_NICKEL_4 := TRUE; END_IF;

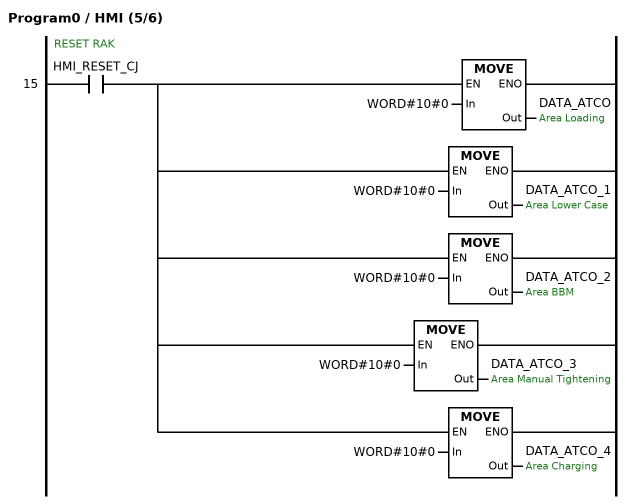
(* Rung 15: RESET RAK *)
IF HMI_RESET_CJ THEN
    DATA_ATCO := WORD#10#0;
    DATA_ATCO_1 := WORD#10#0;
    DATA_ATCO_2 := WORD#10#0;
    DATA_ATCO_3 := WORD#10#0;
    DATA_ATCO_4 := WORD#10#0;
END_IF;

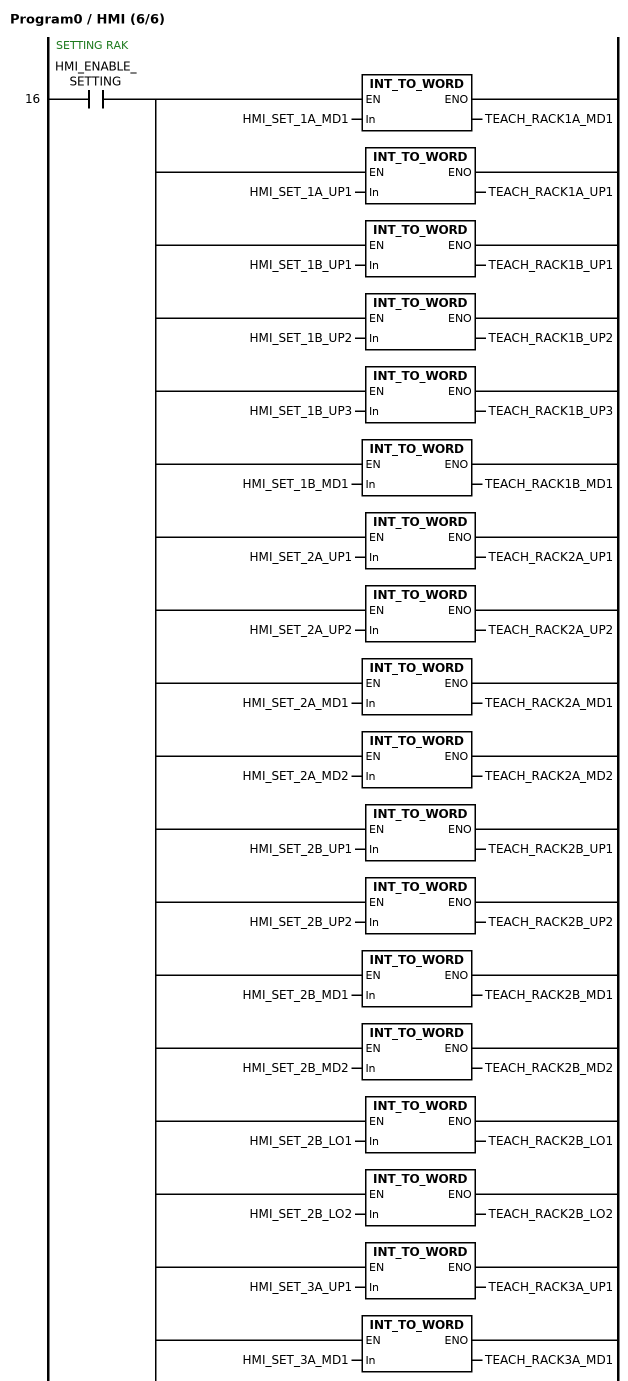

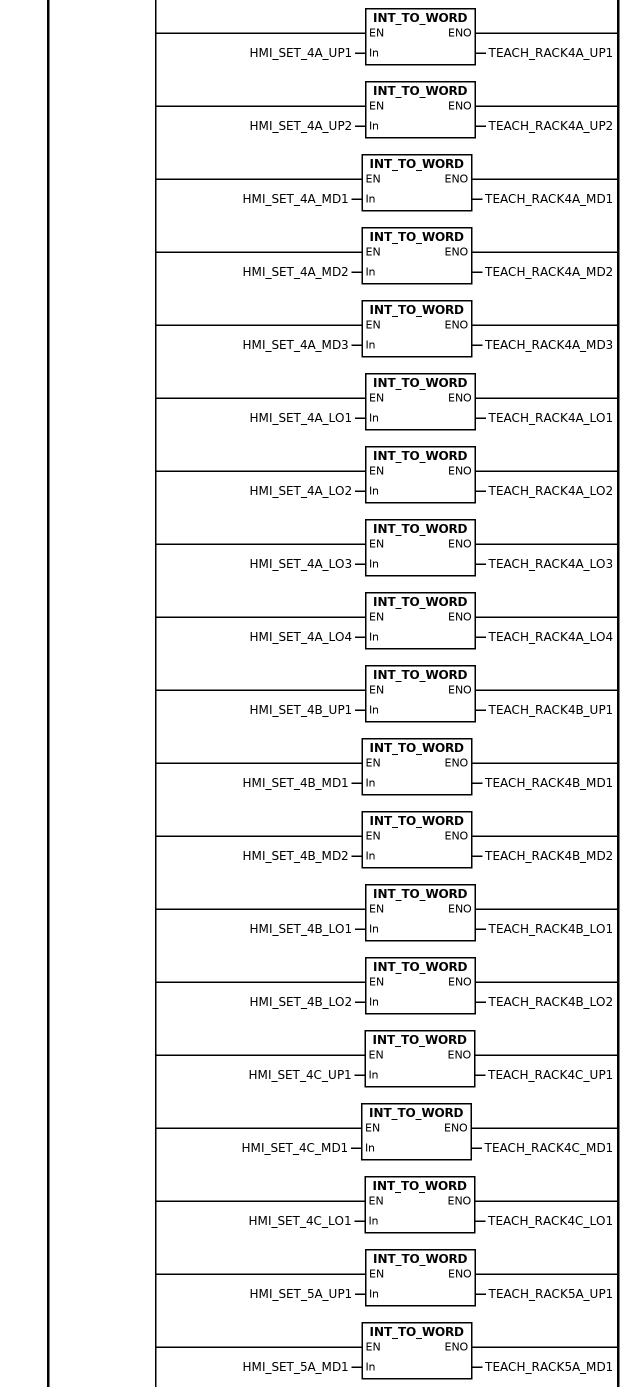

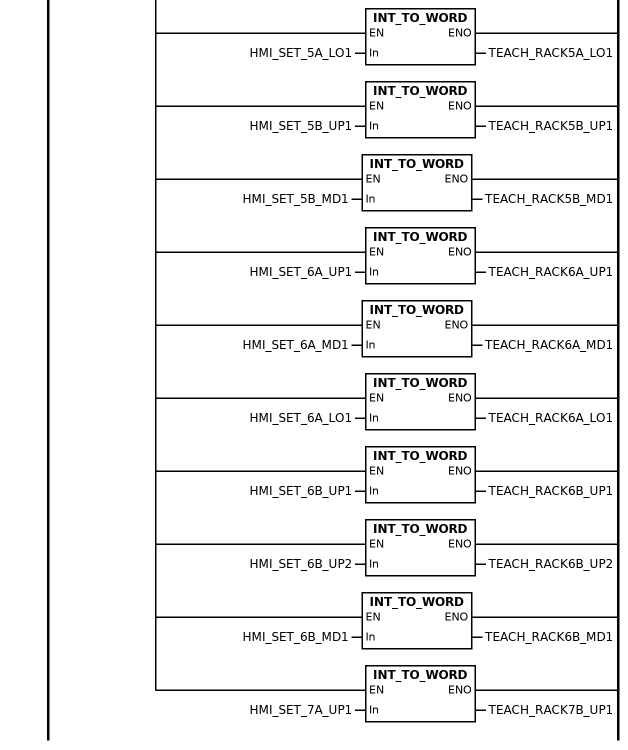
(* Rung 16: SETTING RAK *)
IF HMI_ENABLE_SETTING THEN
    TEACH_RACK1A_MD1 := INT_TO_WORD(In := HMI_SET_1A_MD1);
    TEACH_RACK1A_UP1 := INT_TO_WORD(In := HMI_SET_1A_UP1);
    TEACH_RACK1B_UP1 := INT_TO_WORD(In := HMI_SET_1B_UP1);
    TEACH_RACK1B_UP2 := INT_TO_WORD(In := HMI_SET_1B_UP2);
    TEACH_RACK1B_UP3 := INT_TO_WORD(In := HMI_SET_1B_UP3);
    TEACH_RACK1B_MD1 := INT_TO_WORD(In := HMI_SET_1B_MD1);
    TEACH_RACK2A_UP1 := INT_TO_WORD(In := HMI_SET_2A_UP1);
    TEACH_RACK2A_UP2 := INT_TO_WORD(In := HMI_SET_2A_UP2);
    TEACH_RACK2A_MD1 := INT_TO_WORD(In := HMI_SET_2A_MD1);
    TEACH_RACK2A_MD2 := INT_TO_WORD(In := HMI_SET_2A_MD2);
    TEACH_RACK2B_UP1 := INT_TO_WORD(In := HMI_SET_2B_UP1);
    TEACH_RACK2B_UP2 := INT_TO_WORD(In := HMI_SET_2B_UP2);
    TEACH_RACK2B_MD1 := INT_TO_WORD(In := HMI_SET_2B_MD1);
    TEACH_RACK2B_MD2 := INT_TO_WORD(In := HMI_SET_2B_MD2);
    TEACH_RACK2B_LO1 := INT_TO_WORD(In := HMI_SET_2B_LO1);
    TEACH_RACK2B_LO2 := INT_TO_WORD(In := HMI_SET_2B_LO2);
    TEACH_RACK3A_UP1 := INT_TO_WORD(In := HMI_SET_3A_UP1);
    TEACH_RACK3A_MD1 := INT_TO_WORD(In := HMI_SET_3A_MD1);
    TEACH_RACK4A_UP1 := INT_TO_WORD(In := HMI_SET_4A_UP1);
    TEACH_RACK4A_UP2 := INT_TO_WORD(In := HMI_SET_4A_UP2);
    TEACH_RACK4A_MD1 := INT_TO_WORD(In := HMI_SET_4A_MD1);
    TEACH_RACK4A_MD2 := INT_TO_WORD(In := HMI_SET_4A_MD2);
    TEACH_RACK4A_MD3 := INT_TO_WORD(In := HMI_SET_4A_MD3);
    TEACH_RACK4A_LO1 := INT_TO_WORD(In := HMI_SET_4A_LO1);
    TEACH_RACK4A_LO2 := INT_TO_WORD(In := HMI_SET_4A_LO2);
    TEACH_RACK4A_LO3 := INT_TO_WORD(In := HMI_SET_4A_LO3);
    TEACH_RACK4A_LO4 := INT_TO_WORD(In := HMI_SET_4A_LO4);
    TEACH_RACK4B_UP1 := INT_TO_WORD(In := HMI_SET_4B_UP1);
    TEACH_RACK4B_MD1 := INT_TO_WORD(In := HMI_SET_4B_MD1);
    TEACH_RACK4B_MD2 := INT_TO_WORD(In := HMI_SET_4B_MD2);
    TEACH_RACK4B_LO1 := INT_TO_WORD(In := HMI_SET_4B_LO1);
    TEACH_RACK4B_LO2 := INT_TO_WORD(In := HMI_SET_4B_LO2);
    TEACH_RACK4C_UP1 := INT_TO_WORD(In := HMI_SET_4C_UP1);
    TEACH_RACK4C_MD1 := INT_TO_WORD(In := HMI_SET_4C_MD1);
    TEACH_RACK4C_LO1 := INT_TO_WORD(In := HMI_SET_4C_LO1);
    TEACH_RACK5A_UP1 := INT_TO_WORD(In := HMI_SET_5A_UP1);
    TEACH_RACK5A_MD1 := INT_TO_WORD(In := HMI_SET_5A_MD1);
    TEACH_RACK5A_LO1 := INT_TO_WORD(In := HMI_SET_5A_LO1);
    TEACH_RACK5B_UP1 := INT_TO_WORD(In := HMI_SET_5B_UP1);
    TEACH_RACK5B_MD1 := INT_TO_WORD(In := HMI_SET_5B_MD1);
    TEACH_RACK6A_UP1 := INT_TO_WORD(In := HMI_SET_6A_UP1);
    TEACH_RACK6A_MD1 := INT_TO_WORD(In := HMI_SET_6A_MD1);
    TEACH_RACK6A_LO1 := INT_TO_WORD(In := HMI_SET_6A_LO1);
    TEACH_RACK6B_UP1 := INT_TO_WORD(In := HMI_SET_6B_UP1);
    TEACH_RACK6B_UP2 := INT_TO_WORD(In := HMI_SET_6B_UP2);
    TEACH_RACK6B_MD1 := INT_TO_WORD(In := HMI_SET_6B_MD1);
    TEACH_RACK7B_UP1 := INT_TO_WORD(In := HMI_SET_7A_UP1);
END_IF;

(* Section UDP_ATCO: ladder, written here as Structured Text *)

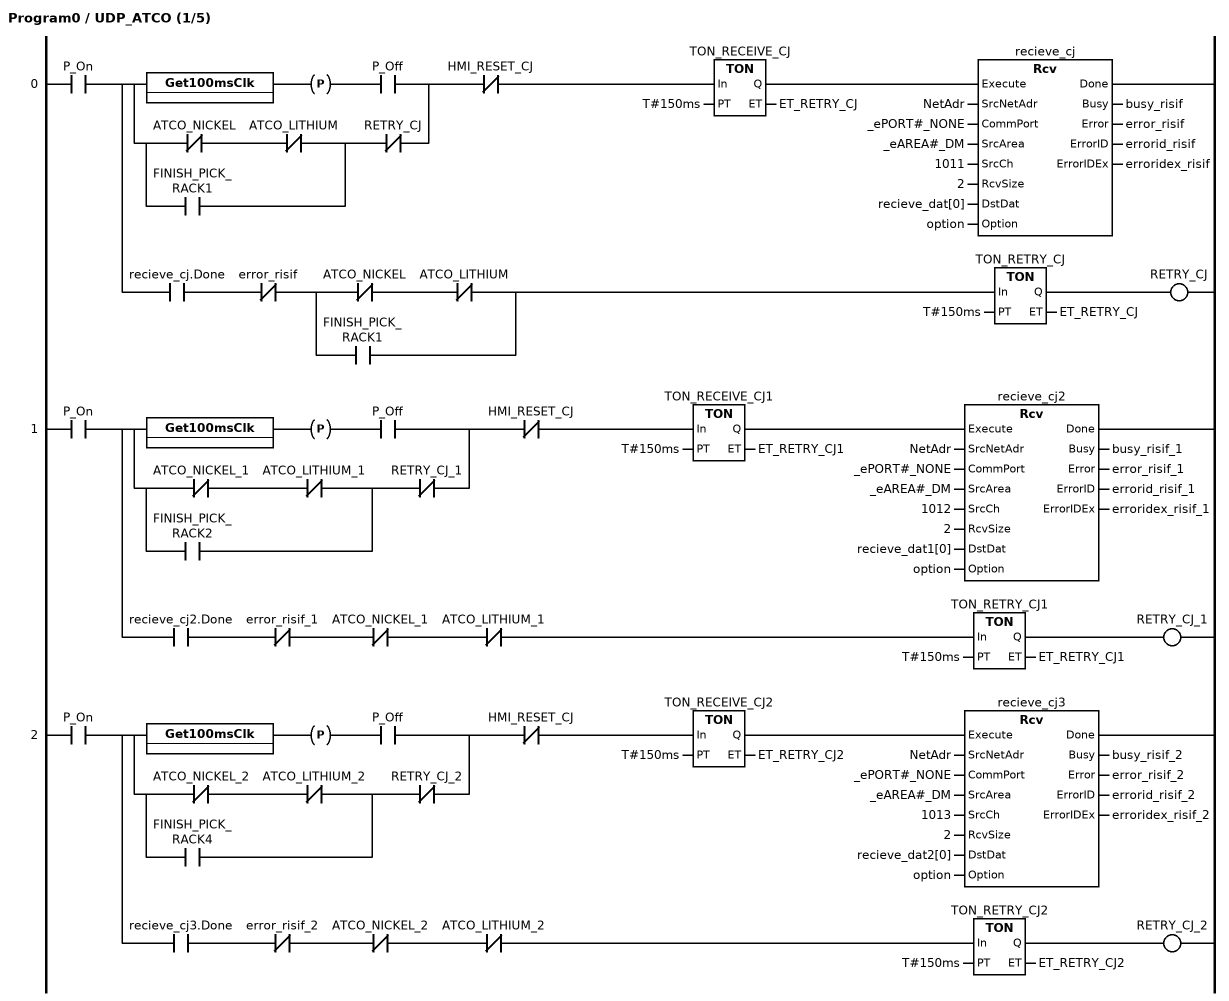
(* Rung 0 *)
_e9(CLK := P_On AND Get100msClk());
TON_RECEIVE_CJ(In := ((_e9.Q AND P_Off) OR (P_On AND ((NOT ATCO_NICKEL AND NOT ATCO_LITHIUM) OR FINISH_PICK_RACK1) AND NOT RETRY_CJ)) AND NOT HMI_RESET_CJ, PT := T#150ms, ET => ET_RETRY_CJ);
recieve_cj(Execute := TON_RECEIVE_CJ.Q, SrcNetAdr := NetAdr, CommPort := _ePORT#_NONE, SrcArea := _eAREA#_DM, SrcCh := 1011, RcvSize := 2, DstDat := recieve_dat[0], Option := option, Busy => busy_risif, Error => error_risif, ErrorID => errorid_risif, ErrorIDEx => erroridex_risif);
TON_RETRY_CJ(In := P_On AND recieve_cj.Done AND NOT error_risif AND ((NOT ATCO_NICKEL AND NOT ATCO_LITHIUM) OR FINISH_PICK_RACK1), PT := T#150ms, ET => ET_RETRY_CJ);
RETRY_CJ := TON_RETRY_CJ.Q;
(* Rung 1 *)
_e10(CLK := P_On AND Get100msClk());
TON_RECEIVE_CJ1(In := ((_e10.Q AND P_Off) OR (P_On AND ((NOT ATCO_NICKEL_1 AND NOT ATCO_LITHIUM_1) OR FINISH_PICK_RACK2) AND NOT RETRY_CJ_1)) AND NOT HMI_RESET_CJ, PT := T#150ms, ET => ET_RETRY_CJ1);
recieve_cj2(Execute := TON_RECEIVE_CJ1.Q, SrcNetAdr := NetAdr, CommPort := _ePORT#_NONE, SrcArea := _eAREA#_DM, SrcCh := 1012, RcvSize := 2, DstDat := recieve_dat1[0], Option := option, Busy => busy_risif_1, Error => error_risif_1, ErrorID => errorid_risif_1, ErrorIDEx => erroridex_risif_1);
TON_RETRY_CJ1(In := P_On AND recieve_cj2.Done AND NOT error_risif_1 AND NOT ATCO_NICKEL_1 AND NOT ATCO_LITHIUM_1, PT := T#150ms, ET => ET_RETRY_CJ1);
RETRY_CJ_1 := TON_RETRY_CJ1.Q;
(* Rung 2 *)
_e11(CLK := P_On AND Get100msClk());
TON_RECEIVE_CJ2(In := ((_e11.Q AND P_Off) OR (P_On AND ((NOT ATCO_NICKEL_2 AND NOT ATCO_LITHIUM_2) OR FINISH_PICK_RACK4) AND NOT RETRY_CJ_2)) AND NOT HMI_RESET_CJ, PT := T#150ms, ET => ET_RETRY_CJ2);
recieve_cj3(Execute := TON_RECEIVE_CJ2.Q, SrcNetAdr := NetAdr, CommPort := _ePORT#_NONE, SrcArea := _eAREA#_DM, SrcCh := 1013, RcvSize := 2, DstDat := recieve_dat2[0], Option := option, Busy => busy_risif_2, Error => error_risif_2, ErrorID => errorid_risif_2, ErrorIDEx => erroridex_risif_2);
TON_RETRY_CJ2(In := P_On AND recieve_cj3.Done AND NOT error_risif_2 AND NOT ATCO_NICKEL_2 AND NOT ATCO_LITHIUM_2, PT := T#150ms, ET => ET_RETRY_CJ2);
RETRY_CJ_2 := TON_RETRY_CJ2.Q;

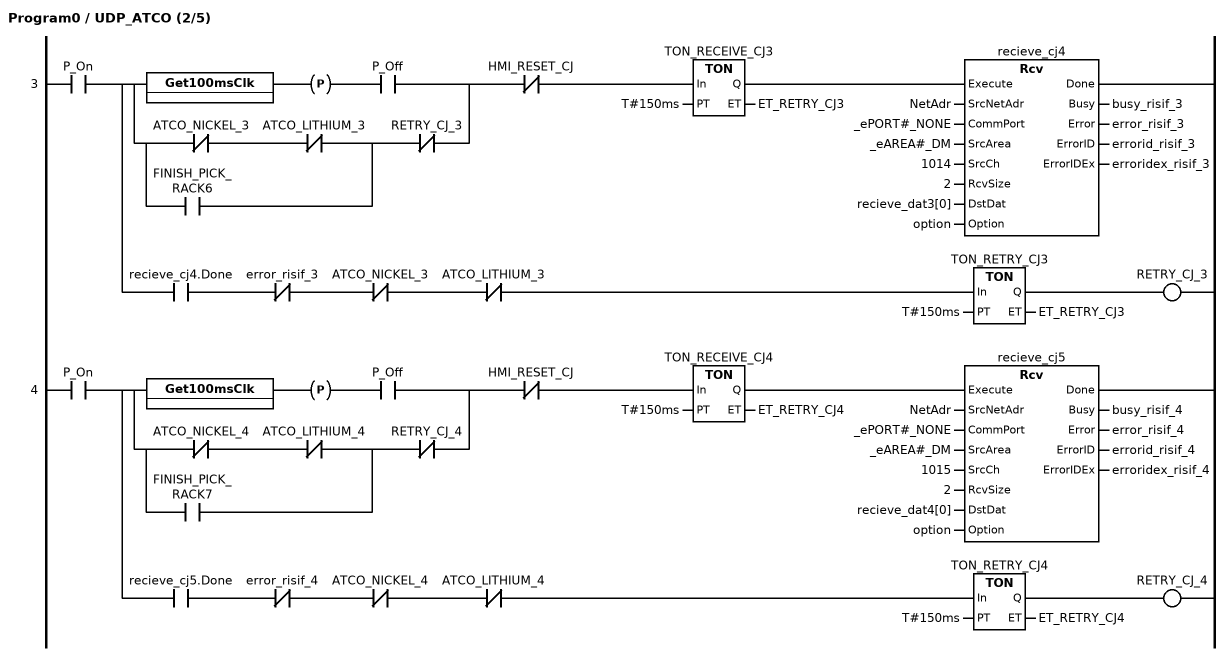
(* Rung 3 *)
_e12(CLK := P_On AND Get100msClk());
TON_RECEIVE_CJ3(In := ((_e12.Q AND P_Off) OR (P_On AND ((NOT ATCO_NICKEL_3 AND NOT ATCO_LITHIUM_3) OR FINISH_PICK_RACK6) AND NOT RETRY_CJ_3)) AND NOT HMI_RESET_CJ, PT := T#150ms, ET => ET_RETRY_CJ3);
recieve_cj4(Execute := TON_RECEIVE_CJ3.Q, SrcNetAdr := NetAdr, CommPort := _ePORT#_NONE, SrcArea := _eAREA#_DM, SrcCh := 1014, RcvSize := 2, DstDat := recieve_dat3[0], Option := option, Busy => busy_risif_3, Error => error_risif_3, ErrorID => errorid_risif_3, ErrorIDEx => erroridex_risif_3);
TON_RETRY_CJ3(In := P_On AND recieve_cj4.Done AND NOT error_risif_3 AND NOT ATCO_NICKEL_3 AND NOT ATCO_LITHIUM_3, PT := T#150ms, ET => ET_RETRY_CJ3);
RETRY_CJ_3 := TON_RETRY_CJ3.Q;
(* Rung 4 *)
_e13(CLK := P_On AND Get100msClk());
TON_RECEIVE_CJ4(In := ((_e13.Q AND P_Off) OR (P_On AND ((NOT ATCO_NICKEL_4 AND NOT ATCO_LITHIUM_4) OR FINISH_PICK_RACK7) AND NOT RETRY_CJ_4)) AND NOT HMI_RESET_CJ, PT := T#150ms, ET => ET_RETRY_CJ4);
recieve_cj5(Execute := TON_RECEIVE_CJ4.Q, SrcNetAdr := NetAdr, CommPort := _ePORT#_NONE, SrcArea := _eAREA#_DM, SrcCh := 1015, RcvSize := 2, DstDat := recieve_dat4[0], Option := option, Busy => busy_risif_4, Error => error_risif_4, ErrorID => errorid_risif_4, ErrorIDEx => erroridex_risif_4);
TON_RETRY_CJ4(In := P_On AND recieve_cj5.Done AND NOT error_risif_4 AND NOT ATCO_NICKEL_4 AND NOT ATCO_LITHIUM_4, PT := T#150ms, ET => ET_RETRY_CJ4);
RETRY_CJ_4 := TON_RETRY_CJ4.Q;

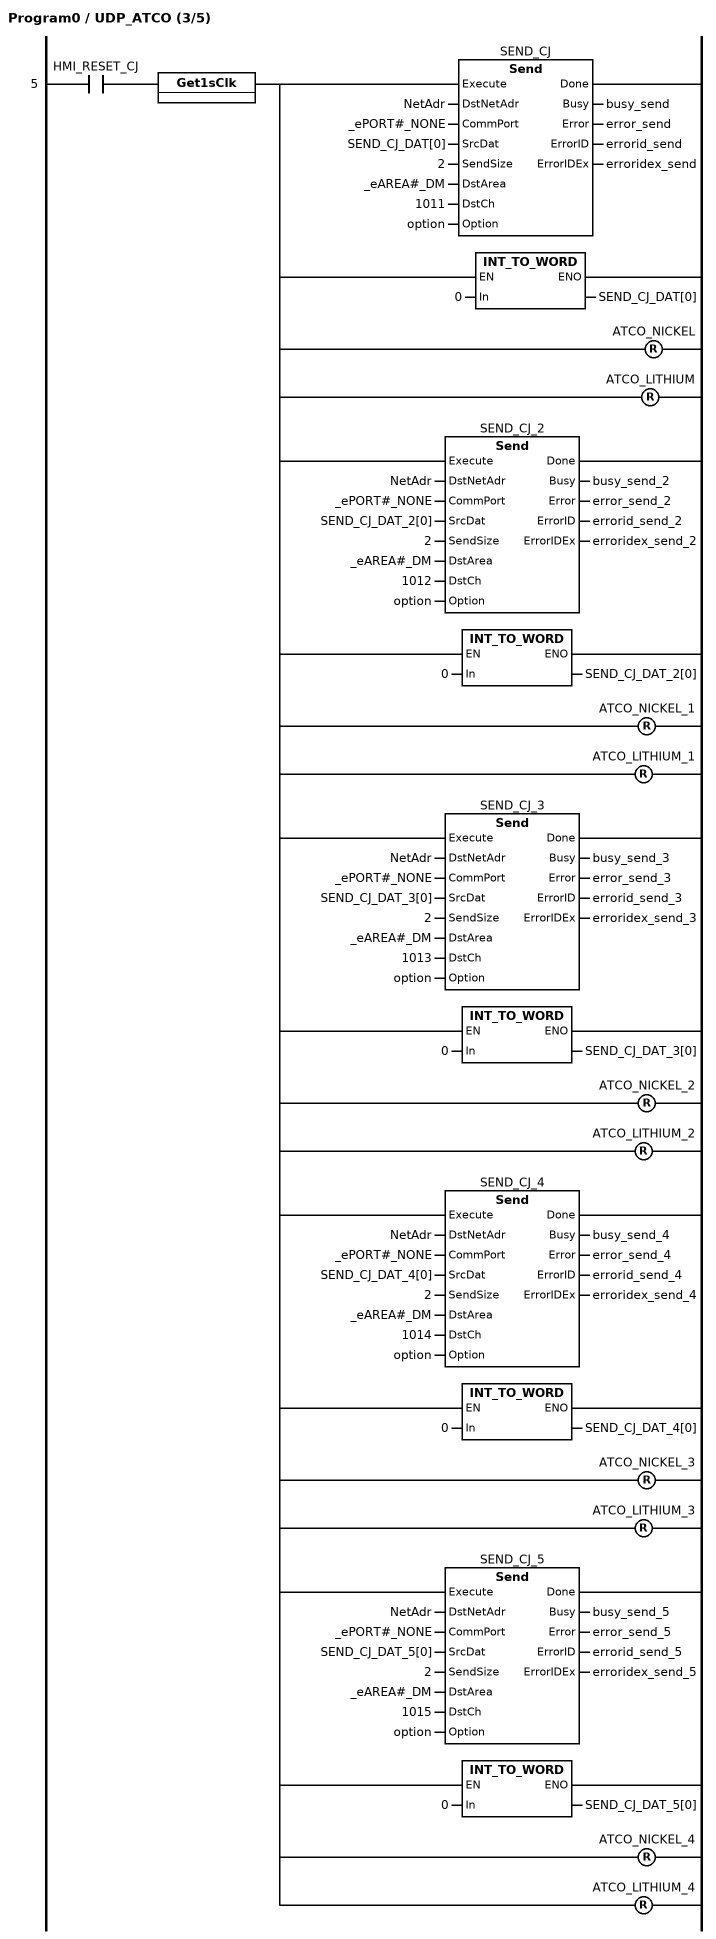
(* Rung 5 *)
SEND_CJ(Execute := HMI_RESET_CJ AND Get1sClk(), DstNetAdr := NetAdr, CommPort := _ePORT#_NONE, SrcDat := SEND_CJ_DAT[0], SendSize := 2, DstArea := _eAREA#_DM, DstCh := 1011, Option := option, Busy => busy_send, Error => error_send, ErrorID => errorid_send, ErrorIDEx => erroridex_send);
IF HMI_RESET_CJ AND Get1sClk() THEN
    SEND_CJ_DAT[0] := INT_TO_WORD(In := 0);
    ATCO_NICKEL := FALSE;
    ATCO_LITHIUM := FALSE;
END_IF;
SEND_CJ_2(Execute := HMI_RESET_CJ AND Get1sClk(), DstNetAdr := NetAdr, CommPort := _ePORT#_NONE, SrcDat := SEND_CJ_DAT_2[0], SendSize := 2, DstArea := _eAREA#_DM, DstCh := 1012, Option := option, Busy => busy_send_2, Error => error_send_2, ErrorID => errorid_send_2, ErrorIDEx => erroridex_send_2);
IF HMI_RESET_CJ AND Get1sClk() THEN
    SEND_CJ_DAT_2[0] := INT_TO_WORD(In := 0);
    ATCO_NICKEL_1 := FALSE;
    ATCO_LITHIUM_1 := FALSE;
END_IF;
SEND_CJ_3(Execute := HMI_RESET_CJ AND Get1sClk(), DstNetAdr := NetAdr, CommPort := _ePORT#_NONE, SrcDat := SEND_CJ_DAT_3[0], SendSize := 2, DstArea := _eAREA#_DM, DstCh := 1013, Option := option, Busy => busy_send_3, Error => error_send_3, ErrorID => errorid_send_3, ErrorIDEx => erroridex_send_3);
IF HMI_RESET_CJ AND Get1sClk() THEN
    SEND_CJ_DAT_3[0] := INT_TO_WORD(In := 0);
    ATCO_NICKEL_2 := FALSE;
    ATCO_LITHIUM_2 := FALSE;
END_IF;
SEND_CJ_4(Execute := HMI_RESET_CJ AND Get1sClk(), DstNetAdr := NetAdr, CommPort := _ePORT#_NONE, SrcDat := SEND_CJ_DAT_4[0], SendSize := 2, DstArea := _eAREA#_DM, DstCh := 1014, Option := option, Busy => busy_send_4, Error => error_send_4, ErrorID => errorid_send_4, ErrorIDEx => erroridex_send_4);
IF HMI_RESET_CJ AND Get1sClk() THEN
    SEND_CJ_DAT_4[0] := INT_TO_WORD(In := 0);
    ATCO_NICKEL_3 := FALSE;
    ATCO_LITHIUM_3 := FALSE;
END_IF;
SEND_CJ_5(Execute := HMI_RESET_CJ AND Get1sClk(), DstNetAdr := NetAdr, CommPort := _ePORT#_NONE, SrcDat := SEND_CJ_DAT_5[0], SendSize := 2, DstArea := _eAREA#_DM, DstCh := 1015, Option := option, Busy => busy_send_5, Error => error_send_5, ErrorID => errorid_send_5, ErrorIDEx => erroridex_send_5);
IF HMI_RESET_CJ AND Get1sClk() THEN
    SEND_CJ_DAT_5[0] := INT_TO_WORD(In := 0);
    ATCO_NICKEL_4 := FALSE;
    ATCO_LITHIUM_4 := FALSE;
END_IF;

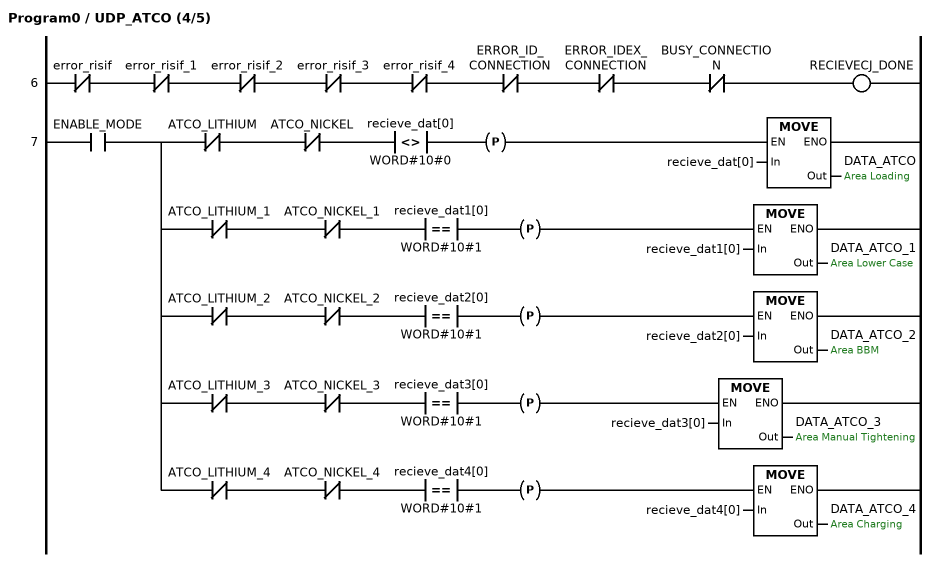
(* Rung 6 *)
RECIEVECJ_DONE := NOT error_risif AND NOT error_risif_1 AND NOT error_risif_2 AND NOT error_risif_3 AND NOT error_risif_4 AND NOT ERROR_ID_CONNECTION AND NOT ERROR_IDEX_CONNECTION AND NOT BUSY_CONNECTION;
(* Rung 7 *)
_e14(CLK := ENABLE_MODE AND NOT ATCO_LITHIUM AND NOT ATCO_NICKEL AND (recieve_dat[0] <> WORD#10#0));
IF _e14.Q THEN DATA_ATCO := recieve_dat[0]; END_IF;
_e15(CLK := ENABLE_MODE AND NOT ATCO_LITHIUM_1 AND NOT ATCO_NICKEL_1 AND (recieve_dat1[0] = WORD#10#1));
IF _e15.Q THEN DATA_ATCO_1 := recieve_dat1[0]; END_IF;
_e16(CLK := ENABLE_MODE AND NOT ATCO_LITHIUM_2 AND NOT ATCO_NICKEL_2 AND (recieve_dat2[0] = WORD#10#1));
IF _e16.Q THEN DATA_ATCO_2 := recieve_dat2[0]; END_IF;
_e17(CLK := ENABLE_MODE AND NOT ATCO_LITHIUM_3 AND NOT ATCO_NICKEL_3 AND (recieve_dat3[0] = WORD#10#1));
IF _e17.Q THEN DATA_ATCO_3 := recieve_dat3[0]; END_IF;
_e18(CLK := ENABLE_MODE AND NOT ATCO_LITHIUM_4 AND NOT ATCO_NICKEL_4 AND (recieve_dat4[0] = WORD#10#1));
IF _e18.Q THEN DATA_ATCO_4 := recieve_dat4[0]; END_IF;

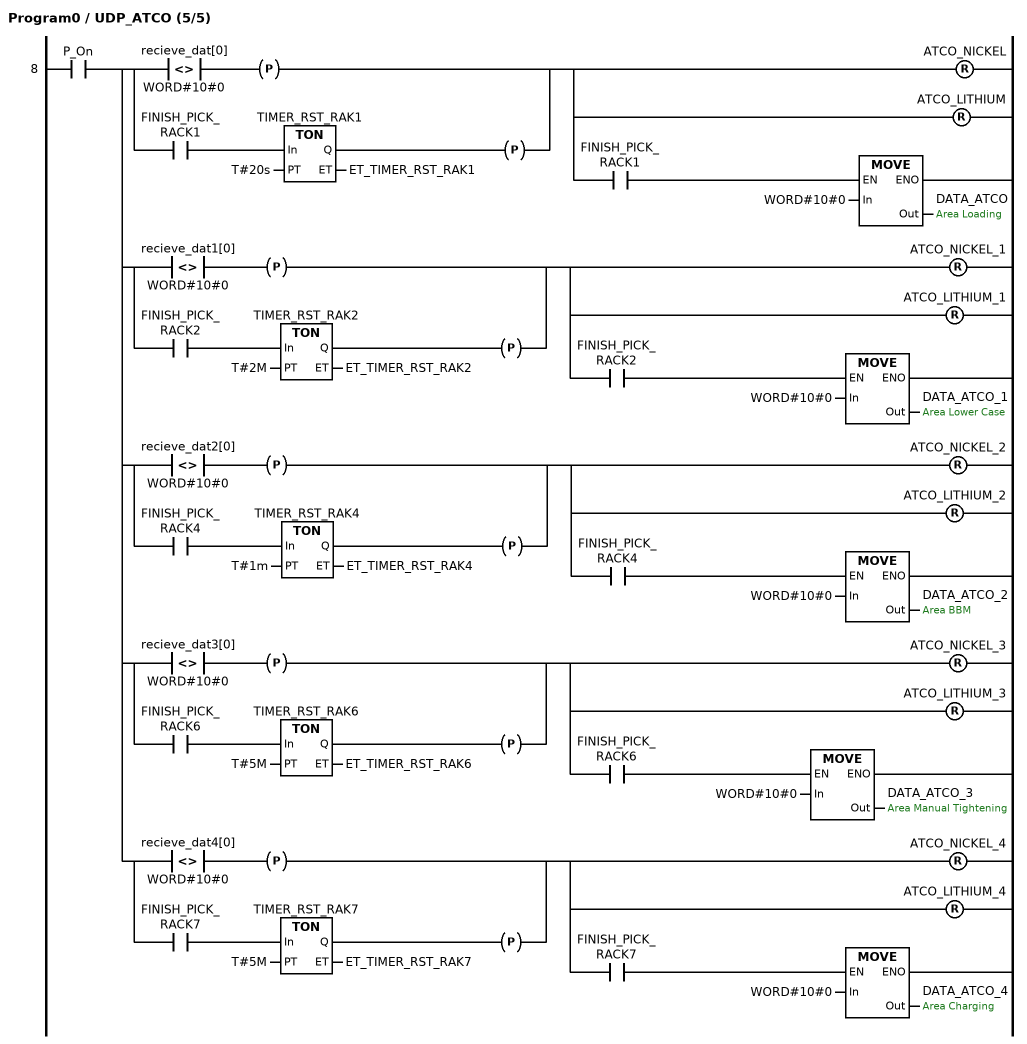
(* Rung 8 *)
_e19(CLK := P_On AND (recieve_dat[0] <> WORD#10#0));
TIMER_RST_RAK1(In := P_On AND FINISH_PICK_RACK1, PT := T#20s, ET => ET_TIMER_RST_RAK1);
_e20(CLK := TIMER_RST_RAK1.Q);
IF _e19.Q OR _e20.Q THEN
    ATCO_NICKEL := FALSE;
    ATCO_LITHIUM := FALSE;
END_IF;
IF (_e19.Q OR _e20.Q) AND FINISH_PICK_RACK1 THEN DATA_ATCO := WORD#10#0; END_IF;
_e21(CLK := P_On AND (recieve_dat1[0] <> WORD#10#0));
TIMER_RST_RAK2(In := P_On AND FINISH_PICK_RACK2, PT := T#2M, ET => ET_TIMER_RST_RAK2);
_e22(CLK := TIMER_RST_RAK2.Q);
IF _e21.Q OR _e22.Q THEN
    ATCO_NICKEL_1 := FALSE;
    ATCO_LITHIUM_1 := FALSE;
END_IF;
IF (_e21.Q OR _e22.Q) AND FINISH_PICK_RACK2 THEN DATA_ATCO_1 := WORD#10#0; END_IF;
_e23(CLK := P_On AND (recieve_dat2[0] <> WORD#10#0));
TIMER_RST_RAK4(In := P_On AND FINISH_PICK_RACK4, PT := T#1m, ET => ET_TIMER_RST_RAK4);
_e24(CLK := TIMER_RST_RAK4.Q);
IF _e23.Q OR _e24.Q THEN
    ATCO_NICKEL_2 := FALSE;
    ATCO_LITHIUM_2 := FALSE;
END_IF;
IF (_e23.Q OR _e24.Q) AND FINISH_PICK_RACK4 THEN DATA_ATCO_2 := WORD#10#0; END_IF;
_e25(CLK := P_On AND (recieve_dat3[0] <> WORD#10#0));
TIMER_RST_RAK6(In := P_On AND FINISH_PICK_RACK6, PT := T#5M, ET => ET_TIMER_RST_RAK6);
_e26(CLK := TIMER_RST_RAK6.Q);
IF _e25.Q OR _e26.Q THEN
    ATCO_NICKEL_3 := FALSE;
    ATCO_LITHIUM_3 := FALSE;
END_IF;
IF (_e25.Q OR _e26.Q) AND FINISH_PICK_RACK6 THEN DATA_ATCO_3 := WORD#10#0; END_IF;
_e27(CLK := P_On AND (recieve_dat4[0] <> WORD#10#0));
TIMER_RST_RAK7(In := P_On AND FINISH_PICK_RACK7, PT := T#5M, ET => ET_TIMER_RST_RAK7);
_e28(CLK := TIMER_RST_RAK7.Q);
IF _e27.Q OR _e28.Q THEN
    ATCO_NICKEL_4 := FALSE;
    ATCO_LITHIUM_4 := FALSE;
END_IF;
IF (_e27.Q OR _e28.Q) AND FINISH_PICK_RACK7 THEN DATA_ATCO_4 := WORD#10#0; END_IF;

(* Section SEQUENCE: ladder, written here as Structured Text *)

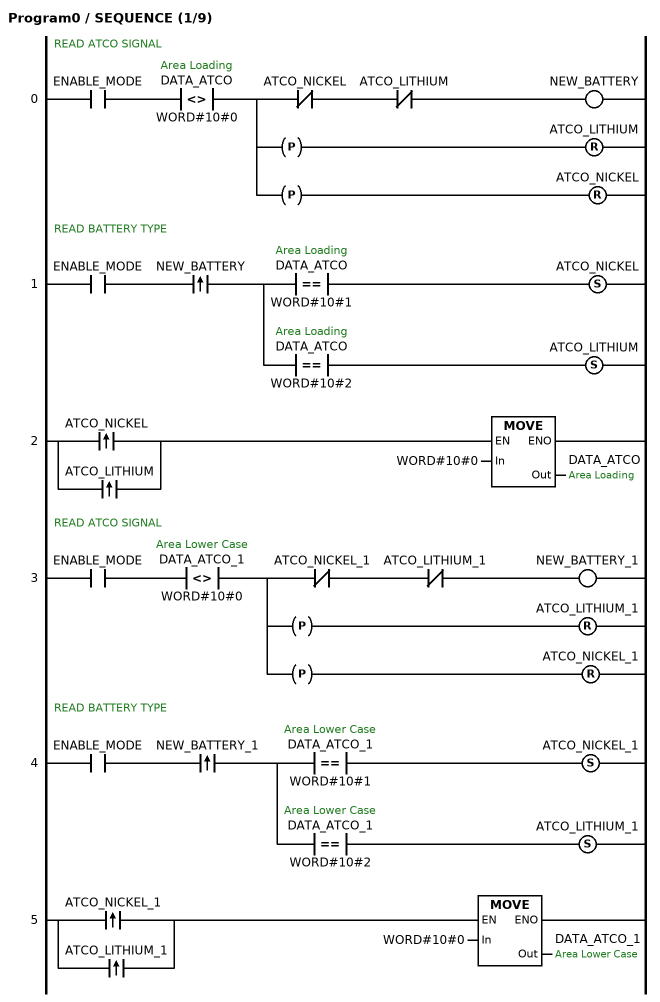
(* Rung 0: READ ATCO SIGNAL *)
NEW_BATTERY := ENABLE_MODE AND (DATA_ATCO <> WORD#10#0) AND NOT ATCO_NICKEL AND NOT ATCO_LITHIUM;
_e29(CLK := ENABLE_MODE AND (DATA_ATCO <> WORD#10#0));
IF _e29.Q THEN ATCO_LITHIUM := FALSE; END_IF;
_e30(CLK := ENABLE_MODE AND (DATA_ATCO <> WORD#10#0));
IF _e30.Q THEN ATCO_NICKEL := FALSE; END_IF;
(* Rung 1: READ BATTERY TYPE *)
_e31(CLK := NEW_BATTERY);
IF ENABLE_MODE AND _e31.Q AND (DATA_ATCO = WORD#10#1) THEN ATCO_NICKEL := TRUE; END_IF;
IF ENABLE_MODE AND _e31.Q AND (DATA_ATCO = WORD#10#2) THEN ATCO_LITHIUM := TRUE; END_IF;
(* Rung 2 *)
_e32(CLK := ATCO_NICKEL);
_e33(CLK := ATCO_LITHIUM);
IF _e32.Q OR _e33.Q THEN DATA_ATCO := WORD#10#0; END_IF;
(* Rung 3: READ ATCO SIGNAL *)
NEW_BATTERY_1 := ENABLE_MODE AND (DATA_ATCO_1 <> WORD#10#0) AND NOT ATCO_NICKEL_1 AND NOT ATCO_LITHIUM_1;
_e34(CLK := ENABLE_MODE AND (DATA_ATCO_1 <> WORD#10#0));
IF _e34.Q THEN ATCO_LITHIUM_1 := FALSE; END_IF;
_e35(CLK := ENABLE_MODE AND (DATA_ATCO_1 <> WORD#10#0));
IF _e35.Q THEN ATCO_NICKEL_1 := FALSE; END_IF;
(* Rung 4: READ BATTERY TYPE *)
_e36(CLK := NEW_BATTERY_1);
IF ENABLE_MODE AND _e36.Q AND (DATA_ATCO_1 = WORD#10#1) THEN ATCO_NICKEL_1 := TRUE; END_IF;
IF ENABLE_MODE AND _e36.Q AND (DATA_ATCO_1 = WORD#10#2) THEN ATCO_LITHIUM_1 := TRUE; END_IF;
(* Rung 5 *)
_e37(CLK := ATCO_NICKEL_1);
_e38(CLK := ATCO_LITHIUM_1);
IF _e37.Q OR _e38.Q THEN DATA_ATCO_1 := WORD#10#0; END_IF;

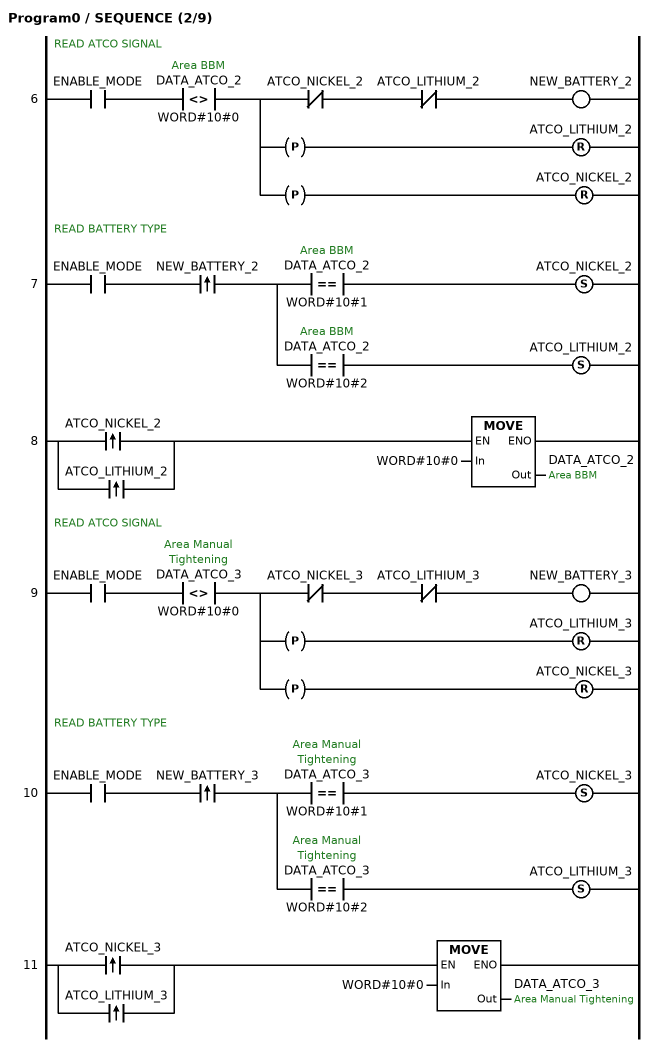
(* Rung 6: READ ATCO SIGNAL *)
NEW_BATTERY_2 := ENABLE_MODE AND (DATA_ATCO_2 <> WORD#10#0) AND NOT ATCO_NICKEL_2 AND NOT ATCO_LITHIUM_2;
_e39(CLK := ENABLE_MODE AND (DATA_ATCO_2 <> WORD#10#0));
IF _e39.Q THEN ATCO_LITHIUM_2 := FALSE; END_IF;
_e40(CLK := ENABLE_MODE AND (DATA_ATCO_2 <> WORD#10#0));
IF _e40.Q THEN ATCO_NICKEL_2 := FALSE; END_IF;
(* Rung 7: READ BATTERY TYPE *)
_e41(CLK := NEW_BATTERY_2);
IF ENABLE_MODE AND _e41.Q AND (DATA_ATCO_2 = WORD#10#1) THEN ATCO_NICKEL_2 := TRUE; END_IF;
IF ENABLE_MODE AND _e41.Q AND (DATA_ATCO_2 = WORD#10#2) THEN ATCO_LITHIUM_2 := TRUE; END_IF;
(* Rung 8 *)
_e42(CLK := ATCO_NICKEL_2);
_e43(CLK := ATCO_LITHIUM_2);
IF _e42.Q OR _e43.Q THEN DATA_ATCO_2 := WORD#10#0; END_IF;
(* Rung 9: READ ATCO SIGNAL *)
NEW_BATTERY_3 := ENABLE_MODE AND (DATA_ATCO_3 <> WORD#10#0) AND NOT ATCO_NICKEL_3 AND NOT ATCO_LITHIUM_3;
_e44(CLK := ENABLE_MODE AND (DATA_ATCO_3 <> WORD#10#0));
IF _e44.Q THEN ATCO_LITHIUM_3 := FALSE; END_IF;
_e45(CLK := ENABLE_MODE AND (DATA_ATCO_3 <> WORD#10#0));
IF _e45.Q THEN ATCO_NICKEL_3 := FALSE; END_IF;
(* Rung 10: READ BATTERY TYPE *)
_e46(CLK := NEW_BATTERY_3);
IF ENABLE_MODE AND _e46.Q AND (DATA_ATCO_3 = WORD#10#1) THEN ATCO_NICKEL_3 := TRUE; END_IF;
IF ENABLE_MODE AND _e46.Q AND (DATA_ATCO_3 = WORD#10#2) THEN ATCO_LITHIUM_3 := TRUE; END_IF;
(* Rung 11 *)
_e47(CLK := ATCO_NICKEL_3);
_e48(CLK := ATCO_LITHIUM_3);
IF _e47.Q OR _e48.Q THEN DATA_ATCO_3 := WORD#10#0; END_IF;

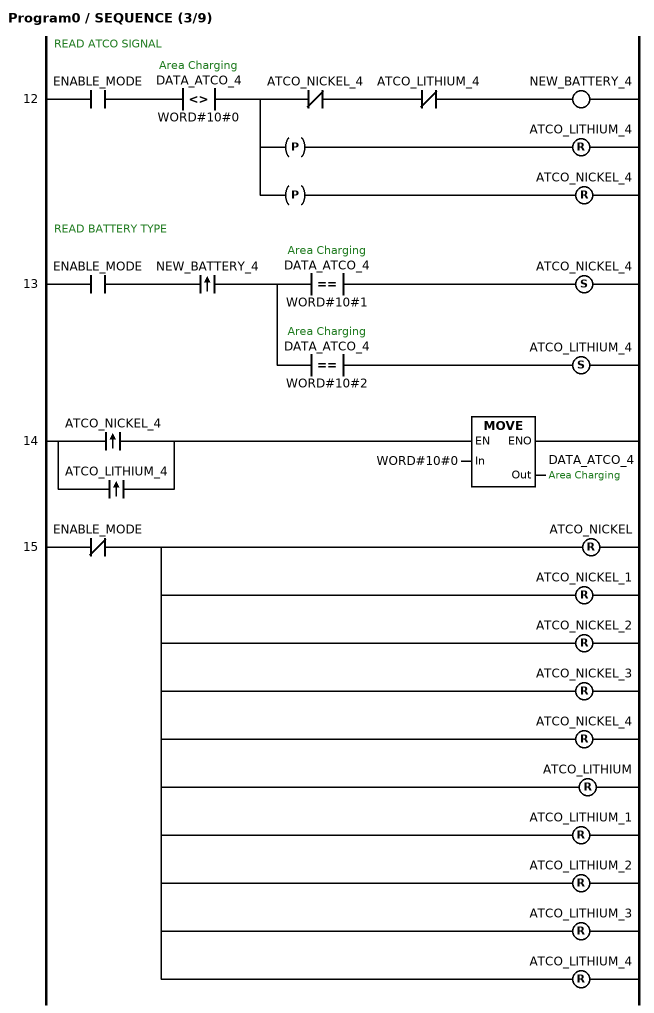
(* Rung 12: READ ATCO SIGNAL *)
NEW_BATTERY_4 := ENABLE_MODE AND (DATA_ATCO_4 <> WORD#10#0) AND NOT ATCO_NICKEL_4 AND NOT ATCO_LITHIUM_4;
_e49(CLK := ENABLE_MODE AND (DATA_ATCO_4 <> WORD#10#0));
IF _e49.Q THEN ATCO_LITHIUM_4 := FALSE; END_IF;
_e50(CLK := ENABLE_MODE AND (DATA_ATCO_4 <> WORD#10#0));
IF _e50.Q THEN ATCO_NICKEL_4 := FALSE; END_IF;
(* Rung 13: READ BATTERY TYPE *)
_e51(CLK := NEW_BATTERY_4);
IF ENABLE_MODE AND _e51.Q AND (DATA_ATCO_4 = WORD#10#1) THEN ATCO_NICKEL_4 := TRUE; END_IF;
IF ENABLE_MODE AND _e51.Q AND (DATA_ATCO_4 = WORD#10#2) THEN ATCO_LITHIUM_4 := TRUE; END_IF;
(* Rung 14 *)
_e52(CLK := ATCO_NICKEL_4);
_e53(CLK := ATCO_LITHIUM_4);
IF _e52.Q OR _e53.Q THEN DATA_ATCO_4 := WORD#10#0; END_IF;
(* Rung 15 *)
IF NOT ENABLE_MODE THEN
    ATCO_NICKEL := FALSE;
    ATCO_NICKEL_1 := FALSE;
    ATCO_NICKEL_2 := FALSE;
    ATCO_NICKEL_3 := FALSE;
    ATCO_NICKEL_4 := FALSE;
    ATCO_LITHIUM := FALSE;
    ATCO_LITHIUM_1 := FALSE;
    ATCO_LITHIUM_2 := FALSE;
    ATCO_LITHIUM_3 := FALSE;
    ATCO_LITHIUM_4 := FALSE;
END_IF;

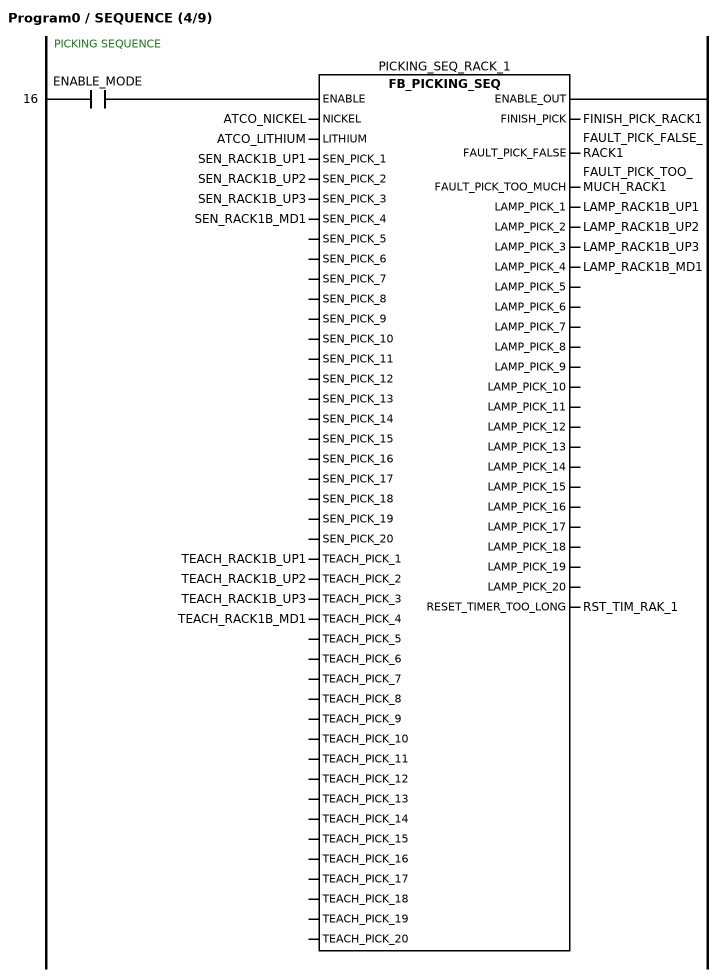
(* Rung 16: PICKING SEQUENCE *)
PICKING_SEQ_RACK_1(ENABLE := ENABLE_MODE, NICKEL := ATCO_NICKEL, LITHIUM := ATCO_LITHIUM, SEN_PICK_1 := SEN_RACK1B_UP1, SEN_PICK_2 := SEN_RACK1B_UP2, SEN_PICK_3 := SEN_RACK1B_UP3, SEN_PICK_4 := SEN_RACK1B_MD1, TEACH_PICK_1 := TEACH_RACK1B_UP1, TEACH_PICK_2 := TEACH_RACK1B_UP2, TEACH_PICK_3 := TEACH_RACK1B_UP3, TEACH_PICK_4 := TEACH_RACK1B_MD1, FINISH_PICK => FINISH_PICK_RACK1, FAULT_PICK_FALSE => FAULT_PICK_FALSE_RACK1, FAULT_PICK_TOO_MUCH => FAULT_PICK_TOO_MUCH_RACK1, LAMP_PICK_1 => LAMP_RACK1B_UP1, LAMP_PICK_2 => LAMP_RACK1B_UP2, LAMP_PICK_3 => LAMP_RACK1B_UP3, LAMP_PICK_4 => LAMP_RACK1B_MD1, RESET_TIMER_TOO_LONG => RST_TIM_RAK_1);

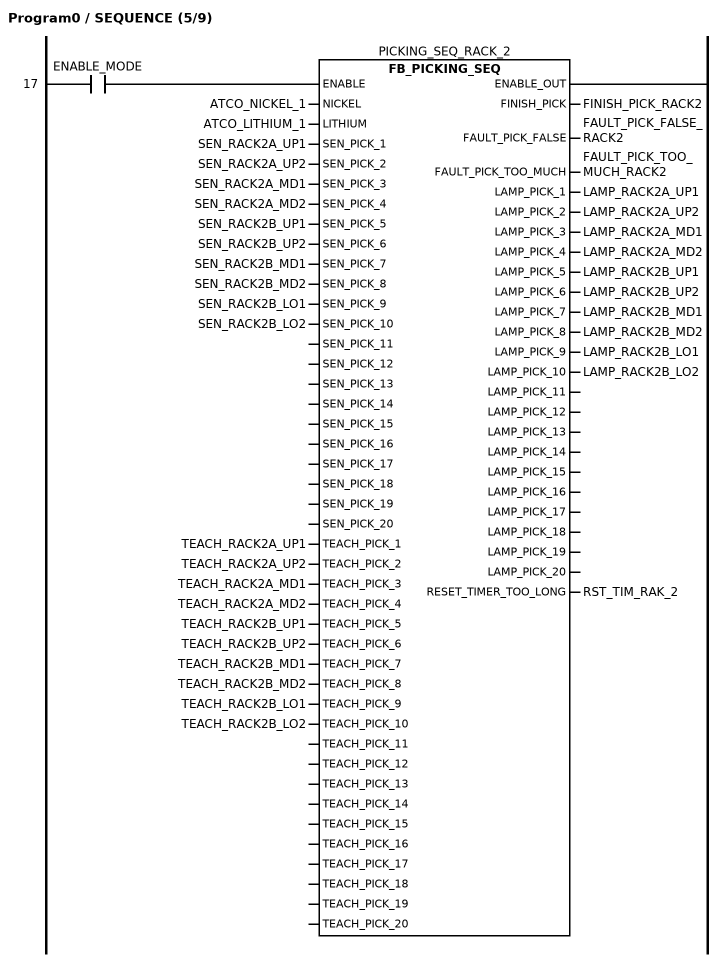
(* Rung 17 *)
PICKING_SEQ_RACK_2(ENABLE := ENABLE_MODE, NICKEL := ATCO_NICKEL_1, LITHIUM := ATCO_LITHIUM_1, SEN_PICK_1 := SEN_RACK2A_UP1, SEN_PICK_2 := SEN_RACK2A_UP2, SEN_PICK_3 := SEN_RACK2A_MD1, SEN_PICK_4 := SEN_RACK2A_MD2, SEN_PICK_5 := SEN_RACK2B_UP1, SEN_PICK_6 := SEN_RACK2B_UP2, SEN_PICK_7 := SEN_RACK2B_MD1, SEN_PICK_8 := SEN_RACK2B_MD2, SEN_PICK_9 := SEN_RACK2B_LO1, SEN_PICK_10 := SEN_RACK2B_LO2, TEACH_PICK_1 := TEACH_RACK2A_UP1, TEACH_PICK_2 := TEACH_RACK2A_UP2, TEACH_PICK_3 := TEACH_RACK2A_MD1, TEACH_PICK_4 := TEACH_RACK2A_MD2, TEACH_PICK_5 := TEACH_RACK2B_UP1, TEACH_PICK_6 := TEACH_RACK2B_UP2, TEACH_PICK_7 := TEACH_RACK2B_MD1, TEACH_PICK_8 := TEACH_RACK2B_MD2, TEACH_PICK_9 := TEACH_RACK2B_LO1, TEACH_PICK_10 := TEACH_RACK2B_LO2, FINISH_PICK => FINISH_PICK_RACK2, FAULT_PICK_FALSE => FAULT_PICK_FALSE_RACK2, FAULT_PICK_TOO_MUCH => FAULT_PICK_TOO_MUCH_RACK2, LAMP_PICK_1 => LAMP_RACK2A_UP1, LAMP_PICK_2 => LAMP_RACK2A_UP2, LAMP_PICK_3 => LAMP_RACK2A_MD1, LAMP_PICK_4 => LAMP_RACK2A_MD2, LAMP_PICK_5 => LAMP_RACK2B_UP1, LAMP_PICK_6 => LAMP_RACK2B_UP2, LAMP_PICK_7 => LAMP_RACK2B_MD1, LAMP_PICK_8 => LAMP_RACK2B_MD2, LAMP_PICK_9 => LAMP_RACK2B_LO1, LAMP_PICK_10 => LAMP_RACK2B_LO2, RESET_TIMER_TOO_LONG => RST_TIM_RAK_2);

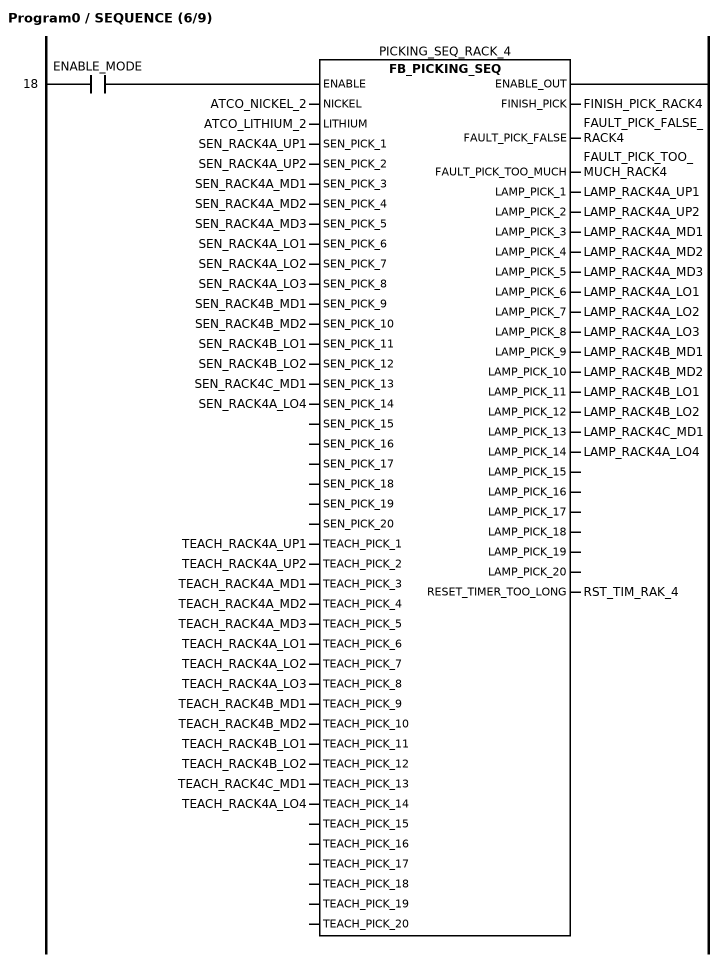
(* Rung 18 *)
PICKING_SEQ_RACK_4(ENABLE := ENABLE_MODE, NICKEL := ATCO_NICKEL_2, LITHIUM := ATCO_LITHIUM_2, SEN_PICK_1 := SEN_RACK4A_UP1, SEN_PICK_2 := SEN_RACK4A_UP2, SEN_PICK_3 := SEN_RACK4A_MD1, SEN_PICK_4 := SEN_RACK4A_MD2, SEN_PICK_5 := SEN_RACK4A_MD3, SEN_PICK_6 := SEN_RACK4A_LO1, SEN_PICK_7 := SEN_RACK4A_LO2, SEN_PICK_8 := SEN_RACK4A_LO3, SEN_PICK_9 := SEN_RACK4B_MD1, SEN_PICK_10 := SEN_RACK4B_MD2, SEN_PICK_11 := SEN_RACK4B_LO1, SEN_PICK_12 := SEN_RACK4B_LO2, SEN_PICK_13 := SEN_RACK4C_MD1, SEN_PICK_14 := SEN_RACK4A_LO4, TEACH_PICK_1 := TEACH_RACK4A_UP1, TEACH_PICK_2 := TEACH_RACK4A_UP2, TEACH_PICK_3 := TEACH_RACK4A_MD1, TEACH_PICK_4 := TEACH_RACK4A_MD2, TEACH_PICK_5 := TEACH_RACK4A_MD3, TEACH_PICK_6 := TEACH_RACK4A_LO1, TEACH_PICK_7 := TEACH_RACK4A_LO2, TEACH_PICK_8 := TEACH_RACK4A_LO3, TEACH_PICK_9 := TEACH_RACK4B_MD1, TEACH_PICK_10 := TEACH_RACK4B_MD2, TEACH_PICK_11 := TEACH_RACK4B_LO1, TEACH_PICK_12 := TEACH_RACK4B_LO2, TEACH_PICK_13 := TEACH_RACK4C_MD1, TEACH_PICK_14 := TEACH_RACK4A_LO4, FINISH_PICK => FINISH_PICK_RACK4, FAULT_PICK_FALSE => FAULT_PICK_FALSE_RACK4, FAULT_PICK_TOO_MUCH => FAULT_PICK_TOO_MUCH_RACK4, LAMP_PICK_1 => LAMP_RACK4A_UP1, LAMP_PICK_2 => LAMP_RACK4A_UP2, LAMP_PICK_3 => LAMP_RACK4A_MD1, LAMP_PICK_4 => LAMP_RACK4A_MD2, LAMP_PICK_5 => LAMP_RACK4A_MD3, LAMP_PICK_6 => LAMP_RACK4A_LO1, LAMP_PICK_7 => LAMP_RACK4A_LO2, LAMP_PICK_8 => LAMP_RACK4A_LO3, LAMP_PICK_9 => LAMP_RACK4B_MD1, LAMP_PICK_10 => LAMP_RACK4B_MD2, LAMP_PICK_11 => LAMP_RACK4B_LO1, LAMP_PICK_12 => LAMP_RACK4B_LO2, LAMP_PICK_13 => LAMP_RACK4C_MD1, LAMP_PICK_14 => LAMP_RACK4A_LO4, RESET_TIMER_TOO_LONG => RST_TIM_RAK_4);

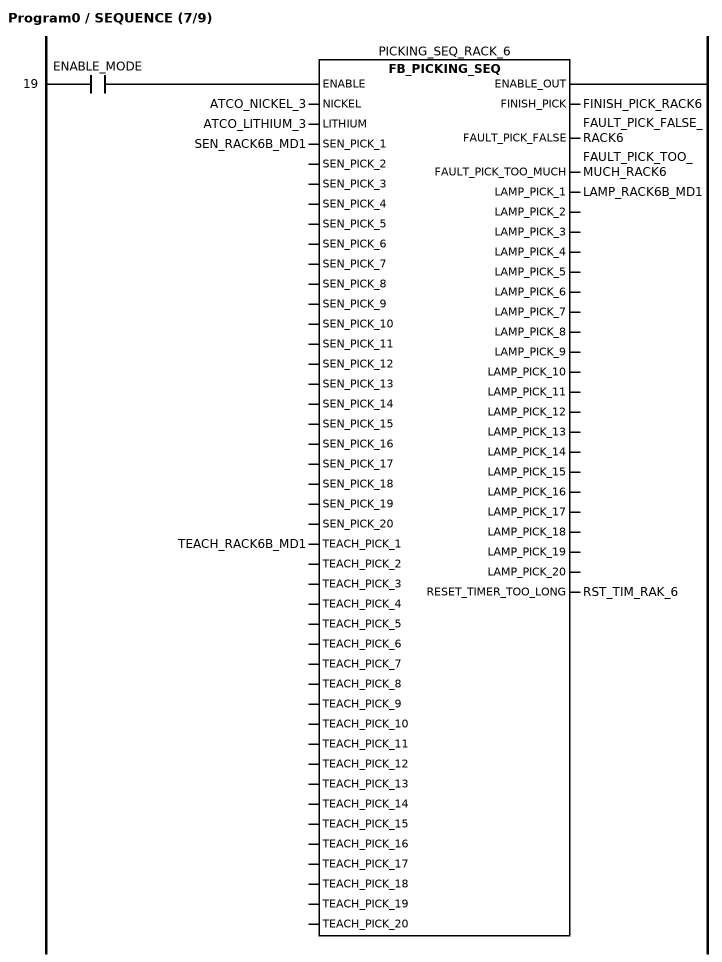
(* Rung 19 *)
PICKING_SEQ_RACK_6(ENABLE := ENABLE_MODE, NICKEL := ATCO_NICKEL_3, LITHIUM := ATCO_LITHIUM_3, SEN_PICK_1 := SEN_RACK6B_MD1, TEACH_PICK_1 := TEACH_RACK6B_MD1, FINISH_PICK => FINISH_PICK_RACK6, FAULT_PICK_FALSE => FAULT_PICK_FALSE_RACK6, FAULT_PICK_TOO_MUCH => FAULT_PICK_TOO_MUCH_RACK6, LAMP_PICK_1 => LAMP_RACK6B_MD1, RESET_TIMER_TOO_LONG => RST_TIM_RAK_6);

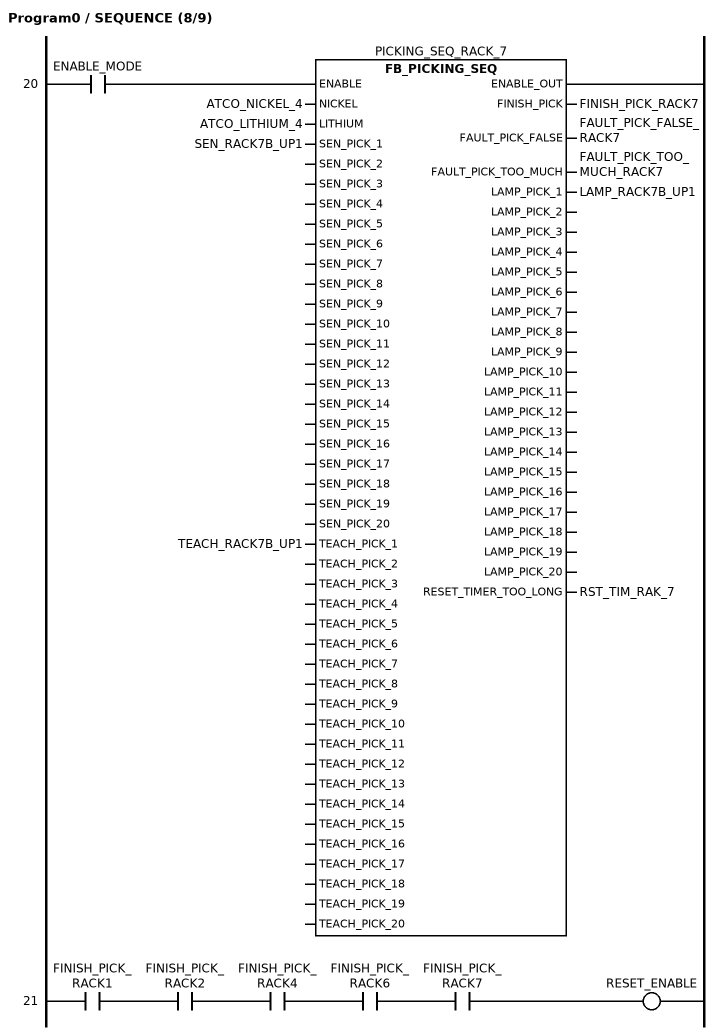
(* Rung 20 *)
PICKING_SEQ_RACK_7(ENABLE := ENABLE_MODE, NICKEL := ATCO_NICKEL_4, LITHIUM := ATCO_LITHIUM_4, SEN_PICK_1 := SEN_RACK7B_UP1, TEACH_PICK_1 := TEACH_RACK7B_UP1, FINISH_PICK => FINISH_PICK_RACK7, FAULT_PICK_FALSE => FAULT_PICK_FALSE_RACK7, FAULT_PICK_TOO_MUCH => FAULT_PICK_TOO_MUCH_RACK7, LAMP_PICK_1 => LAMP_RACK7B_UP1, RESET_TIMER_TOO_LONG => RST_TIM_RAK_7);
(* Rung 21 *)
RESET_ENABLE := FINISH_PICK_RACK1 AND FINISH_PICK_RACK2 AND FINISH_PICK_RACK4 AND FINISH_PICK_RACK6 AND FINISH_PICK_RACK7;

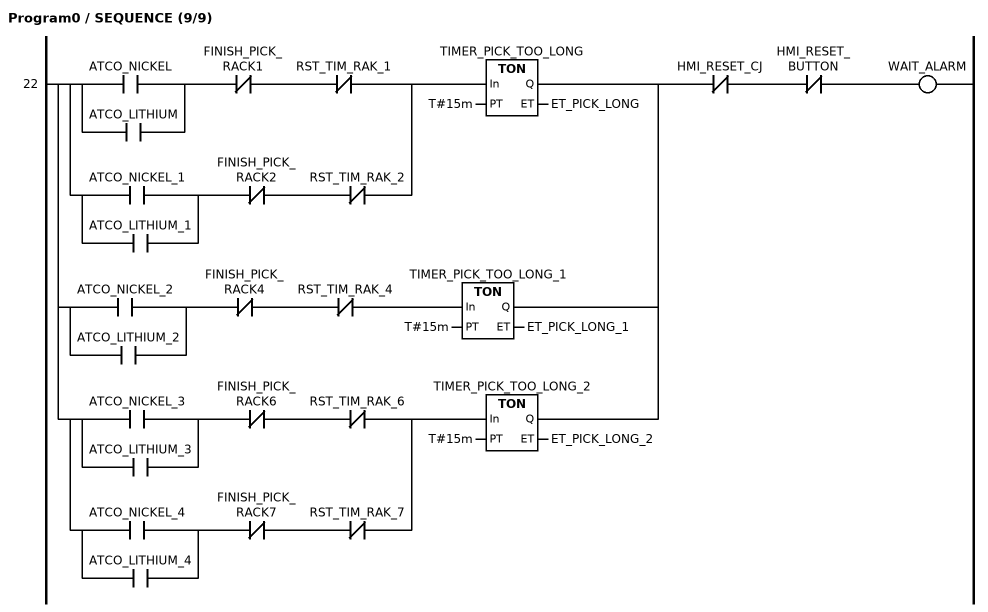
(* Rung 22 *)
TIMER_PICK_TOO_LONG(In := ((ATCO_NICKEL OR ATCO_LITHIUM) AND NOT FINISH_PICK_RACK1 AND NOT RST_TIM_RAK_1) OR ((ATCO_NICKEL_1 OR ATCO_LITHIUM_1) AND NOT FINISH_PICK_RACK2 AND NOT RST_TIM_RAK_2), PT := T#15m, ET => ET_PICK_LONG);
TIMER_PICK_TOO_LONG_1(In := (ATCO_NICKEL_2 OR ATCO_LITHIUM_2) AND NOT FINISH_PICK_RACK4 AND NOT RST_TIM_RAK_4, PT := T#15m, ET => ET_PICK_LONG_1);
TIMER_PICK_TOO_LONG_2(In := ((ATCO_NICKEL_3 OR ATCO_LITHIUM_3) AND NOT FINISH_PICK_RACK6 AND NOT RST_TIM_RAK_6) OR ((ATCO_NICKEL_4 OR ATCO_LITHIUM_4) AND NOT FINISH_PICK_RACK7 AND NOT RST_TIM_RAK_7), PT := T#15m, ET => ET_PICK_LONG_2);
WAIT_ALARM := (TIMER_PICK_TOO_LONG.Q OR TIMER_PICK_TOO_LONG_1.Q OR TIMER_PICK_TOO_LONG_2.Q) AND NOT HMI_RESET_CJ AND NOT HMI_RESET_BUTTON;

(* Section INPUT: ladder, written here as Structured Text *)

